// TIA Portal V17 program export: 3 tag tables, 0 data types, 10 data blocks, 17 code blocks (in call order from the OBs), 11 instance data blocks

VAR_GLOBAL   // PLC tag table "ALARMES"
   ALM0 AT %MW100 : Word;   // ALARMES MB-01
   ALM2 AT %MW102 : Word;   // ALARMES MB-02
   ALM4 AT %MW104 : Word;   // ALARMES MB-03
   ALM6 AT %MW106 : Word;   // ALARMES MB-04
   ALM8 AT %MW108 : Word;   // ALARMES LIT_001
   ALM10 AT %MW110 : Word;   // ALARMES PCM-EEE
   ALM12 AT %MW112 : Word;   // ALARMES QGBT
   ALM14 AT %MW114 : Word;   // ALARMES CHAVE DE NIVEL
   ALM16 AT %MW116 : Word;   // ALARMES PCE-EEE
END_VAR

VAR_GLOBAL   // PLC tag table "Default tag table"
   System_Byte AT %MB1 : Byte;
   FirstScan AT %M1.0 : Bool;
   DiagStatusUpdate AT %M1.1 : Bool;
   AlwaysTRUE AT %M1.2 : Bool;
   AlwaysFALSE AT %M1.3 : Bool;
   Clock_Byte AT %MB0 : Byte;
   Clock_10Hz AT %M0.0 : Bool;
   Clock_5Hz AT %M0.1 : Bool;
   "Clock_2.5Hz" AT %M0.2 : Bool;
   Clock_2Hz AT %M0.3 : Bool;
   "Clock_1.25Hz" AT %M0.4 : Bool;
   Clock_1Hz AT %M0.5 : Bool;
   "Clock_0.625Hz" AT %M0.6 : Bool;
   "Clock_0.5Hz" AT %M0.7 : Bool;
   Tag_3 AT %M50.0 : Bool;
   bloqueio_provisorio AT %M2.0 : Bool;
   pause AT %M2.1 : Bool;
   bloqueio_provisorio_1 AT %M2.2 : Bool;
   Tag_4 AT %M83.0 : Bool;
   CON_MOD AT %MW80 : Int;
   INI AT %M82.0 : Bool;
END_VAR

VAR_GLOBAL   // PLC tag table "IO"
   PCM_EEE_EMER AT %I0.0 : Bool;   // PCM-E-CF-01-04 BOTAO DE EMERGENCIA - ATUADO
   PCM_EEE_K27 AT %I0.1 : Bool;   // PCM-E-CF-01-04 RELE DE PROTECAO FUNCAO 27 - ATUADO
   PCM_EEE_DJL AT %I0.2 : Bool;   // PCM-E-CF-01-04 DISJUNTOR GERAL STATUS - LIGADO
   PCM_EEE_DJD AT %I0.3 : Bool;   // PCM-E-CF-01-04 DISJUNTOR GERAL STATUS - DESLIGADO
   PCM_EEE_DJYFAL AT %I0.4 : Bool;   // PCM-E-CF-01-04 DISJUNTOR GERAL STATUS - FALHA
   PCM_EEE_DJFG AT %I0.5 : Bool;   // PCM-E-CF-01-04 FALHA GERAL ATUADO
   PCM_EEE_TR01_KA3 AT %I0.6 : Bool;   // PCM-E-CF-01-04 TRANSFORMADOR -TR-01 ALARME TEMP 150°
   PCM_EEE_TR01_KA4 AT %I0.7 : Bool;   // PCM-E-CF-01-04 TRANSFORMADOR -TR-01 ALARME TEMP 155°
   PCM_EEE_TR01_KA5 AT %I1.0 : Bool;   // PCM-E-CF-01-04 TRANSFORMADOR -TR-01 FALHA PROTECAO
   PCM_EEE_INTRU AT %I1.1 : Bool;   // PCM-E-CF-01-04 INTRUSAO NO PAINEL (COLUNA 01~04)
   MB_01_FF AT %I1.2 : Bool;   // MB-01 FALTA DE FASE
   MB_01_MMNT AT %I1.3 : Bool;   // MB-01 MODO MANUTENCAO
   MB_01_ML AT %I1.4 : Bool;   // MB-01 MODO LOCAL
   MB_01_MA AT %I1.5 : Bool;   // MB-01 MODO AUTOMATICO
   MB_01_MN AT %I1.6 : Bool;   // MB-01 MODO NORMAL
   MB_01_HMNT AT %I1.7 : Bool;   // MB-01 HABILITA MANUTENCAO
   MB_01_BL AT %I2.0 : Bool;   // MB-01 BOMBA LIGADA
   MB_01_DINV AT %I2.1 : Bool;   // MB-01 DEFEITO NO INVERSOR
   MB_01_DMB AT %I2.2 : Bool;   // MB-01 DEFEITO NA BOMBA
   MB_01_RST AT %I2.3 : Bool;   // MB-01 RESET
   MB_01_INTRU AT %I2.4 : Bool;   // MB-01 INTRUSAO NO PAINEL
   MB_01_EMER AT %I2.5 : Bool;   // MB-01 EMERGENCIA
   MB_02_FF AT %I2.6 : Bool;   // MB-02 FALTA DE FASE
   MB_02_MMNT AT %I2.7 : Bool;   // MB-02 MODO MANUTENCAO
   MB_02_ML AT %I3.0 : Bool;   // MB-02 MODO LOCAL
   MB_02_MA AT %I3.1 : Bool;   // MB-02 MODO AUTOMATICO
   MB_02_MN AT %I3.2 : Bool;   // MB-02 MODO NORMAL
   MB_02_HMNT AT %I3.3 : Bool;   // MB-02 HABILITA MANUTENCAO
   MB_02_BL AT %I3.4 : Bool;   // MB-02 BOMBA LIGADA
   MB_02_DINV AT %I3.5 : Bool;   // MB-02 DEFEITO NO INVERSOR
   MB_02_DMB AT %I3.6 : Bool;   // MB-02 DEFEITO NA BOMBA
   MB_02_RST AT %I3.7 : Bool;   // MB-02 RESET
   MB_02_INTRU AT %I4.0 : Bool;   // MB-02 INTRUSAO NO PAINEL
   MB_02_EMER AT %I4.1 : Bool;   // MB-02 EMERGENCIA
   MB_03_FF AT %I4.2 : Bool;   // MB-03 FALTA DE FASE
   MB_03_MMNT AT %I4.3 : Bool;   // MB-03 MODO MANUTENCAO
   MB_03_ML AT %I4.4 : Bool;   // MB-03 MODO LOCAL
   MB_03_MA AT %I4.5 : Bool;   // MB-03 MODO AUTOMATICO
   MB_03_MN AT %I4.6 : Bool;   // MB-03 MODO NORMAL
   MB_03_HMNT AT %I4.7 : Bool;   // MB-03 HABILITA MANUTENCAO
   MB_03_BL AT %I5.0 : Bool;   // MB-03 BOMBA LIGADA
   MB_03_DINV AT %I5.1 : Bool;   // MB-03 DEFEITO NO INVERSOR
   MB_03_DMB AT %I5.2 : Bool;   // MB-03 DEFEITO NA BOMBA
   MB_03_RST AT %I5.3 : Bool;   // MB-03 RESET
   MB_03_INTRU AT %I5.4 : Bool;   // MB-03 INTRUSAO NO PAINEL
   MB_03_EMER AT %I5.5 : Bool;   // MB-03EMERGENCIA
   MB_04_FF AT %I5.6 : Bool;   // MB-04 FALTA DE FASE
   MB_04_MMNT AT %I5.7 : Bool;   // MB-04 MODO MANUTENCAO
   MB_04_ML AT %I6.0 : Bool;   // MB-04 MODO LOCAL
   MB_04_MA AT %I6.1 : Bool;   // MB-04 MODO AUTOMATICO
   MB_04_MN AT %I6.2 : Bool;   // MB-04 MODO NORMAL
   MB_04_HMNT AT %I6.3 : Bool;   // MB-04 HABILITA MANUTENCAO
   MB_04_BL AT %I6.4 : Bool;   // MB-04 BOMBA LIGADA
   MB_04_DINV AT %I6.5 : Bool;   // MB-04 DEFEITO NO INVERSOR
   MB_04_DMB AT %I6.6 : Bool;   // MB-04 DEFEITO NA BOMBA
   MB_04_RST AT %I6.7 : Bool;   // MB-04 RESET
   MB_04_INTRU AT %I7.0 : Bool;   // MB-04 INTRUSAO NO PAINEL
   MB_04_EMER AT %I7.1 : Bool;   // MB-04 EMERGENCIA
   QGBT_EMER AT %I7.2 : Bool;   // QGBT-AUX-01 BOTAO DE EMERGENCIA ATUADO
   QGBT_K27 AT %I7.3 : Bool;   // QGBT-AUX-01 RELE DE PROTECAO FUNCAO 27/59 ATUADO
   QGBT_DISJ_LIG AT %I7.4 : Bool;   // QGBT-AUX-01 DISJUNTOR GERAL STATUS - LIGADO
   QGBT_DISJ_DESLIG AT %I7.5 : Bool;   // QGBT-AUX-01 DISJUNTOR GERAL STATUS - DESLIGADO
   QGBT_DISJ_YFAL AT %I7.6 : Bool;   // QGBT-AUX-01 DISJUNTOR GERAL FALHA - TRIP
   QGBT_INTRU AT %I7.7 : Bool;   // QGBT-AUX-01 INTRUSAO NO PAINEL
   KI165 AT %I8.0 : Bool;   // RESERVA
   KI166 AT %I8.1 : Bool;   // RESERVA
   KI167 AT %I8.2 : Bool;   // RESERVA
   KI168 AT %I8.3 : Bool;   // RESERVA
   KI169 AT %I8.4 : Bool;   // RESERVA
   KI170 AT %I8.5 : Bool;   // RESERVA
   KI171 AT %I8.6 : Bool;   // RESERVA
   KI172 AT %I8.7 : Bool;   // RESERVA
   LSL_001 AT %I9.0 : Bool;   // CHAVE DE NIVEL -LSL-001
   LSH_001 AT %I9.1 : Bool;   // CHAVE DE NIVEL -LSH-001
   LSL_002 AT %I9.2 : Bool;   // CHAVE DE NIVEL -LSL-002
   LSH_002 AT %I9.3 : Bool;   // CHAVE DE NIVEL -LSH-002
   PCE_EEE_INTRU AT %I9.4 : Bool;   // INTRUSAO NO PAINEL
   PCE_EEE_UPS_ALM AT %I9.5 : Bool;   // UPS EM ALARME FALHA NA BATERIA
   PCE_EEE_UPS_FE AT %I9.6 : Bool;   // UPS EM OPERACAO FALTA DE ENERGIA
   PCE_EEE_UPS_CHAR AT %I9.7 : Bool;   // UPS EM ALARME BATERIA CARREGADA
   MB_01_SH AT %Q0.0 : Bool;   // MB-01 SOLICITACAO HIDRAULICA
   MB_01_PH AT %Q0.1 : Bool;   // MB-01 PROTECAO HIDRAULICA
   MB_01_INTV AT %Q0.2 : Bool;   // MB-01 INTERVALO (COM)
   MB_01_RR AT %Q0.3 : Bool;   // MB-01 RESET REMOTO
   MB_01_INTVS AT %Q0.4 : Bool;   // MB-01 INTERVALO SINAL
   MB_02_SH AT %Q0.5 : Bool;   // MB-02 SOLICITACAO HIDRAULICA
   MB_02_PH AT %Q0.6 : Bool;   // MB-02 PROTECAO HIDRAULICA
   MB_02_INTV AT %Q0.7 : Bool;   // MB-02 INTERVALO (COM)
   MB_02_RR AT %Q1.0 : Bool;   // MB-02 RESET REMOTO
   MB_02_INTVS AT %Q1.1 : Bool;   // MB-02 INTERVALO SINAL
   MB_03_SH AT %Q1.2 : Bool;   // MB-03 SOLICITACAO HIDRAULICA
   MB_03_PH AT %Q1.3 : Bool;   // MB-03 PROTECAO HIDRAULICA
   MB_03_INTV AT %Q1.4 : Bool;   // MB-03 INTERVALO (COM)
   MB_03_RR AT %Q1.5 : Bool;   // MB-03 RESET REMOTO
   MB_03_INTVS AT %Q1.6 : Bool;   // MB-03 INTERVALO SINAL
   MB_04_SH AT %Q1.7 : Bool;   // MB-04 SOLICITACAO HIDRAULICA
   LIT_001 AT %IW10 : Int;   // -LIT-001 TRANSMISSOR DE NIVEL TANQUE (TIPO RADAR)
   MB_01_REF_VEL AT %IW12 : Int;   // REFERENCIA DE VELOCIDADE INVERSOR DE FREQUENCIA BOMBA 01
   MB_02_REF_VEL AT %IW14 : Int;   // REFERENCIA DE VELOCIDADE INVERSOR DE FREQUENCIA BOMBA 02
   MB_03_REF_VEL AT %IW16 : Int;   // REFERENCIA DE VELOCIDADE INVERSOR DE FREQUENCIA BOMBA 03
   MB_04_REF_VEL AT %IW18 : Int;   // REFERENCIA DE VELOCIDADE INVERSOR DE FREQUENCIA BOMBA 04
   FB6 AT %IW20 : Int;   // RESERVA
   FB7 AT %IW22 : Int;   // RESERVA
   FB8 AT %IW24 : Int;   // RESERVA
   FB9 AT %IW26 : Int;   // RESERVA
   FB10 AT %IW28 : Int;   // RESERVA
   FB11 AT %IW30 : Int;   // RESERVA
   FB12 AT %IW32 : Int;   // RESERVA
   FB13 AT %IW34 : Int;   // RESERVA
   FB14 AT %IW36 : Int;   // RESERVA
   FB15 AT %IW38 : Int;   // RESERVA
   FB16 AT %IW40 : Int;   // RESERVA
   MB_01_VEL AT %QW4 : Int;   // SETPOINT INVERSOR DE FREQUENCIA BOMBA 01
   MB_02_VEL AT %QW6 : Int;   // SETPOINT INVERSOR DE FREQUENCIA BOMBA 02
   MB_03_VEL AT %QW8 : Int;   // SETPOINT INVERSOR DE FREQUENCIA BOMBA 03
   MB_04_VEL AT %QW10 : Int;   // SETPOINT INVERSOR DE FREQUENCIA BOMBA 04
   F25 AT %QW12 : Int;   // RESERVA
   F26 AT %QW14 : Int;   // RESERVA
   F27 AT %QW16 : Int;   // RESERVA
   F28 AT %QW18 : Int;   // RESERVA
   MB_04_PH AT %Q2.0 : Bool;   // MB-04 PROTECAO HIDRAULICA
   MB_04_INTV AT %Q2.1 : Bool;   // MB-04 INTERVALO (COM)
   MB_04_RR AT %Q2.2 : Bool;   // MB-04 RESET REMOTO
   MB_04_INTVS AT %Q2.3 : Bool;   // MB-04 INTERVALO SINAL
   KO21 AT %Q2.4 : Bool;   // RESERVA
   KO22 AT %Q2.5 : Bool;   // RESERVA
   KO23 AT %Q2.6 : Bool;   // RESERVA
   KO24 AT %Q2.7 : Bool;   // RESERVA
   KO25 AT %Q3.0 : Bool;   // RESERVA
   KO26 AT %Q3.1 : Bool;   // RESERVA
   KO27 AT %Q3.2 : Bool;   // RESERVA
   KO28 AT %Q3.3 : Bool;   // RESERVA
   KO29 AT %Q3.4 : Bool;   // RESERVA
   KO30 AT %Q3.5 : Bool;   // RESERVA
   KO31 AT %Q3.6 : Bool;   // RESERVA
   KO32 AT %Q3.7 : Bool;   // RESERVA
END_VAR

DATA_BLOCK "ALARMES"   // DB301
{ S7_Optimized_Access := 'TRUE' }
VERSION : 0.1
// stored: AutoNumber false, DBAccessibleFromOPCUA true, IsOnlyStoredInLoadMemory false, IsRetainMemResEnabled false, IsWriteProtectedInAS false, MemoryReserve 100
   VAR
      "CCM-02-EA-P100-YFC" : Bool;   // Falha de comunicação com medidor do CCM1
      "CCM-02-EB-P100-YFC" : Bool;   // Falha de comunicação com medidor do CCM2
      "LIT_001-YHH" : Bool;   // Alarme de nível muito alto do tanque água bruta
      "LIT_001-YH" : Bool;   // Alarme de nível alto do tanque água bruta
      "LIT_001-YL" : Bool;   // Alarme de nível baixo do tanque água bruta
      "LIT_001-YLL" : Bool;   // Alarme de nível muito baixo do tanque água bruta
      "LIT_001-YFS" : Bool;   // Transmissor de nível do tanque água bruta com falha de sinal
      "LIT_001-YHHH" : Bool;   // Alarme de nível muito alto - desliga CAB e lavagem peneira
      "CAB-PT-015-YH" : Bool;
      "CAB-PT-015-YFS" : Bool;
      "MB-03-YIP" : Bool;   // MB-03 com intervalo entre partidas
      "MB-02-YIP" : Bool;   // MB-02 com intervalo entre partidas
      "MB-01-YIP" : Bool;   // MB-01 com intervalo entre partidas
   END_VAR
BEGIN
END_DATA_BLOCK

DATA_BLOCK "COMANDOS"   // DB303
{ S7_Optimized_Access := 'FALSE' }
VERSION : 0.1
// stored: AutoNumber false, DBAccessibleFromOPCUA true, IsOnlyStoredInLoadMemory false, IsWriteProtectedInAS false
   VAR RETAIN
      "MB-01-HS9" : Bool := false;   // Comando disponível
      "MB-01-HS10" : Bool := false;   // Comando disponível
      "MB-01-HS11" : Bool;   // Comando disponível
      "MB-01-HS12" : Bool;   // Comando disponível
      "MB-01-HS13" : Bool;   // Comando disponível
      "MB-01-HS14" : Bool;   // Comando disponível
      "MB-01-HS15" : Bool;   // Comando disponível
      "MB-01-HS16" : Bool;   // Comando disponível
      "MB-01-HS1" : Bool := true;   // Comando manual/automático
      "MB-01-HS2" : Bool := false;   // Comando liga
      "MB-01-HS3" : Bool := false;   // Comando desliga
      "MB-01-HS4" : Bool := false;   // Comando reset falha
      "MB-01-HS5" : Bool := false;   // Comando reset tempo de operação
      "MB-01-HS6" : Bool;
      "MB-01-HS7" : Bool := false;   // Comando habilita bloqueio
      "MB-01-HS8" : Bool := false;   // Comando disponível
      "MB-02-HS9" : Bool := false;   // Comando disponível
      "MB-02-HS10" : Bool := false;   // Comando disponível
      "MB-02-HS11" : Bool;   // Comando disponível
      "MB-02-HS12" : Bool;   // Comando disponível
      "MB-02-HS13" : Bool;   // Comando disponível
      "MB-02-HS14" : Bool;   // Comando disponível
      "MB-02-HS15" : Bool;   // Comando disponível
      "MB-02-HS16" : Bool;   // Comando disponível
      "MB-02-HS1" : Bool := true;   // Comando manual/automático
      "MB-02-HS2" : Bool := false;   // Comando liga
      "MB-02-HS3" : Bool := false;   // Comando desliga
      "MB-02-HS4" : Bool := false;   // Comando reset falha
      "MB-02-HS5" : Bool := false;   // Comando reset tempo de operação
      "MB-02-HS6" : Bool;
      "MB-02-HS7" : Bool := false;   // Comando habilita bloqueio
      "MB-02-HS8" : Bool := false;   // Comando disponível
      "MB-03-HS9" : Bool := false;   // Comando disponível
      "MB-03-HS10" : Bool := false;   // Comando disponível
      "MB-03-HS11" : Bool;   // Comando disponível
      "MB-03-HS12" : Bool;   // Comando disponível
      "MB-03-HS13" : Bool;   // Comando disponível
      "MB-03-HS14" : Bool;   // Comando disponível
      "MB-03-HS15" : Bool;   // Comando disponível
      "MB-03-HS16" : Bool;   // Comando disponível
      "MB-03-HS1" : Bool := true;   // Comando manual/automático
      "MB-03-HS2" : Bool := false;   // Comando liga
      "MB-03-HS3" : Bool := false;   // Comando desliga
      "MB-03-HS4" : Bool := false;   // Comando reset falha
      "MB-03-HS5" : Bool := false;   // Comando reset tempo de operação
      "MB-03-HS6" : Bool;
      "MB-03-HS7" : Bool := false;   // Comando habilita bloqueio
      "MB-03-HS8" : Bool := false;   // Comando disponível
      "MB-04-HS9" : Bool := false;   // Comando disponível
      "MB-04-HS10" : Bool := false;   // Comando disponível
      "MB-04-HS11" : Bool;   // Comando disponível
      "MB-04-HS12" : Bool;   // Comando disponível
      "MB-04-HS13" : Bool;   // Comando disponível
      "MB-04-HS14" : Bool;   // Comando disponível
      "MB-04-HS15" : Bool;   // Comando disponível
      "MB-04-HS16" : Bool;   // Comando disponível
      "MB-04-HS1" : Bool := false;   // Comando manual/automático
      "MB-04-HS2" : Bool := false;   // Comando liga
      "MB-04-HS3" : Bool := false;   // Comando desliga
      "MB-04-HS4" : Bool := false;   // Comando reset falha
      "MB-04-HS5" : Bool := false;   // Comando reset tempo de operação
      "MB-04-HS6" : Bool;
      "MB-04-HS7" : Bool := false;   // Comando habilita bloqueio
      "MB-04-HS8" : Bool := false;   // Comando disponível
      "LIT_001-HS9" : Bool;   // Comando disponível
      "LIT_001-HS10" : Bool;   // Comando disponível
      "LIT_001-HS11" : Bool;   // Comando disponível
      "LIT_001-HS12" : Bool;   // Comando disponível
      "LIT_001-HS13" : Bool;   // Comando disponível
      "LIT_001-HS14" : Bool;   // Comando disponível
      "LIT_001-HS15" : Bool;   // Comando disponível
      "LIT_001-HS16" : Bool;   // Comando disponível
      "LIT_001-HSHH" : Bool;   // Inibe alarme muito alto montante peneira 1
      "LIT_001-HSH" : Bool;   // Inibe alarme nível alto montante peneira 1
      "LIT_001-HSL" : Bool;   // Inibe alarme nível baixo montante peneira 1
      "LIT_001-HSLL" : Bool;   // Inibe alarme nível muito baixo montante peneira 1
      "LIT_001-HSM" : Bool;   // Habilita valor manual para medidor
      "LIT_001-HS6" : Bool;   // Comando disponível
      "LIT_001-HS7" : Bool;   // Comando disponível
      "LIT_001-HS8" : Bool;   // Comando disponível
      "PID-TA3-HI" : Bool;   // Habilita integrall PID tanque de aeração
      "PID-EEEB-HD" : Bool;   // Habilita derivativo PID tanque de aeração
      "PID-EEEB-HP" : Bool;   // Habilita proporcional PID tanque de aeração
      "PID-EEEB-HI" : Bool;   // Habilita integrall PID tanque de aeração
      "PID-TA5-HD" : Bool;   // Habilita derivativo PID tanque de aeração
      "PID-TA5-HP" : Bool;   // Habilita proporcional PID tanque de aeração
      "PID-TA5-HI" : Bool;   // Habilita integrall PID tanque de aeração
      "PID-TA1-HM" : Bool;   // Habilita valor manual para saída
      "PID-TA1-HD" : Bool;   // Habilita derivativo PID tanque de aeração
      "PID-TA1-HP" : Bool;   // Habilita proporcional PID tanque de aeração
      "PID-TA1-HI" : Bool;   // Habilita integrall PID tanque de aeração
      "PID-TA2-HD" : Bool;   // Habilita derivativo PID tanque de aeração
      "PID-TA2-HP" : Bool;   // Habilita proporcional PID tanque de aeração
      "PID-TA2-HI" : Bool;   // Habilita integrall PID tanque de aeração
      "PID-TA3-HD" : Bool;   // Habilita derivativo PID tanque de aeração
      "PID-TA3-HP" : Bool;   // Habilita proporcional PID tanque de aeração
      "PID-TA2-HM" : Bool;   // Habilita valor manual para saída
      "PID-TA3-HM" : Bool;   // Habilita valor manual para saída
      "PID-EEEB-HM" : Bool;   // Habilita valor manual para saída
      "PID-TA5-HM" : Bool;   // Habilita valor manual para saída
   END_VAR
BEGIN
END_DATA_BLOCK

DATA_BLOCK "DIVERSOS"   // DB1
{ S7_Optimized_Access := 'TRUE' }
VERSION : 0.1
// stored: AutoNumber false, DBAccessibleFromOPCUA true, IsOnlyStoredInLoadMemory false, IsRetainMemResEnabled false, IsWriteProtectedInAS false, MemoryReserve 100
   VAR
      T1S : Bool;   // PULSO A CADA 1 SEGUNDO
      AUX_T1S : Bool;   // PULSO A CADA 1 SEGUNDO
      QTDE_PULSO : DInt := 200;
      ForcePulso : Bool;
      N_L00P : Int;
      Aux_N_LOOP : Int;
      Looping : Int := 0;
      TMR : Array[0..10] of IEC_TIMER;
      P1S { S7_SetPoint := 'True'} : Bool;   // Pulso de 1 segundo
      "MB-01-SP" : Bool;   // Solicitação partida de bomba
      "MB-02-SP" : Bool;   // Solicitação partida de bomba
      "MB-03-SP" : Bool;   // Solicitação partida de bomba
      "MB-04-SP" : Bool;   // Solicitação partida de bomba
   END_VAR
BEGIN
END_DATA_BLOCK

DATA_BLOCK "Digitais"   // DB300
{ S7_Optimized_Access := 'FALSE' }
VERSION : 0.1
// stored: AutoNumber false, DBAccessibleFromOPCUA true, IsOnlyStoredInLoadMemory false, IsWriteProtectedInAS false
   VAR RETAIN
      "MB-01-YSH" : Bool;   // Elevatoria principal 1 ligado
      "MB-01-YR" : Bool;   // Elevatoria principal 1 remoto
      "MB-01-YF" : Bool;   // Elevatoria principal 1 falha
      "MB-01-YFF" : Bool;   // Elevatoria principal 1 falta de fase
      "MB-01-MM" : Bool;   // Elevatoria principal 1 modo manutenção
      "MB-01-MA" : Bool;   // Elevatoria principal 1 modo automatico
      "MB-01-EMER" : Bool;   // Elevatoria principal 1 emergencia
      "MB-01-MN" : Bool;   // Elevatoria principal 1 modo normal
      "MB-01-ML" : Bool;   // Elevatoria principal 1 modo local
      "MB-01-YFI" : Bool;   // Elevatoria principal 1 com falha no inversor
      "MB-01-YFA" : Bool;   // Elevatoria principal 1 com falha no acionamento
      "MB-01-YPTA" : Bool;   // Elevatoria principal 1 com proteção térmica atuada
      "MB-01-HM" : Bool;   // Elevatoria principal 1 habilita manutenção
      "MB-01-RST" : Bool;   // Elevatoria principal 1 reset
      "MB-01-INTRU" : Bool;   // Elevatoria principal 1 intrusão no painel
      "MB-01-YFB" : Bool;   // Elevatoria principal 1 defeito na bomba
      "MB-02-YSH" : Bool;   // Elevatoria principal 2 ligado
      "MB-02-YR" : Bool;   // Elevatoria principal 2 remoto
      "MB-02-YF" : Bool;   // Elevatoria principal 2 falha
      "MB-02-YFF" : Bool;   // Elevatoria principal 2 falta de fase
      "MB-02-MM" : Bool;   // Elevatoria principal 2 modo manutenção
      "MB-02-MA" : Bool;   // Elevatoria principal 2 modo automatico
      "MB-02-EMER" : Bool;   // Elevatoria principal 2 emergencia
      "MB-02-MN" : Bool;   // Elevatoria principal 2 modo normal
      "MB-02-ML" : Bool;   // Elevatoria principal 2 modo local
      "MB-02-YFI" : Bool;   // Elevatoria principal 2 com falha no inversor
      "MB-02-YFA" : Bool;   // Elevatoria principal 2 com falha no acionamento
      "MB-02-YPTA" : Bool;   // Elevatoria principal 2 com proteção térmica atuada
      "MB-02-HM" : Bool;   // Elevatoria principal 2 habilita manutenção
      "MB-02-RST" : Bool;   // Elevatoria principal 2 reset
      "MB-02-INTRU" : Bool;   // Elevatoria principal 2 intrusão no painel
      "MB-02-YFB" : Bool;   // Elevatoria principal 2 defeito na bomba
      "MB-03-YSH" : Bool;   // Elevatoria principal 3 ligado
      "MB-03-YR" : Bool;   // Elevatoria principal 3 remoto
      "MB-03-YF" : Bool;   // Elevatoria principal 3 falha
      "MB-03-YFF" : Bool;   // Elevatoria principal 3 falta de fase
      "MB-03-MM" : Bool;   // Elevatoria principal 3 modo manutenção
      "MB-03-MA" : Bool;   // Elevatoria principal 3 modo automatico
      "MB-03-EMER" : Bool;   // Elevatoria principal 3 emergencia
      "MB-03-MN" : Bool;   // Elevatoria principal 3 modo normal
      "MB-03-ML" : Bool;   // Elevatoria principal 3 modo local
      "MB-03-YFI" : Bool;   // Elevatoria principal 3 com falha no inversor
      "MB-03-YFA" : Bool;   // Elevatoria principal 3 com falha no acionamento
      "MB-03-YPTA" : Bool;   // Elevatoria principal 3 com proteção térmica atuada
      "MB-03-HM" : Bool;   // Elevatoria principal 3 habilita manutenção
      "MB-03-RST" : Bool;   // Elevatoria principal 3 reset
      "MB-03-INTRU" : Bool;   // Elevatoria principal 3 intrusão no painel
      "MB-03-YFB" : Bool;   // Elevatoria principal 3 defeito na bomba
      "MB-04-YSH" : Bool;   // Elevatoria principal 4 ligado
      "MB-04-YR" : Bool;   // Elevatoria principal 4 remoto
      "MB-04-YF" : Bool;   // Elevatoria principal 4 falha
      "MB-04-YFF" : Bool;   // Elevatoria principal 4 falta de fase
      "MB-04-MM" : Bool;   // Elevatoria principal 4 modo manutenção
      "MB-04-MA" : Bool;   // Elevatoria principal 4 modo automatico
      "MB-04-EMER" : Bool;   // Elevatoria principal 4 emergencia
      "MB-04-MN" : Bool;   // Elevatoria principal 4 modo normal
      "MB-04-ML" : Bool;   // Elevatoria principal 4 modo local
      "MB-04-YFI" : Bool;   // Elevatoria principal 4 com falha no inversor
      "MB-04-YFA" : Bool;   // Elevatoria principal 4 com falha no acionamento
      "MB-04-YPTA" : Bool;   // Elevatoria principal 4 com proteção térmica atuada
      "MB-04-HM" : Bool;   // Elevatoria principal 4 habilita manutenção
      "MB-04-RST" : Bool;   // Elevatoria principal 4 reset
      "MB-04-INTRU" : Bool;   // Elevatoria principal 4 intrusão no painel
      "MB-04-YFB" : Bool;   // Elevatoria principal 4 defeito na bomba
      "LIT_001-AL8" : Bool;   // Disponível para alarme
      "LIT_001-AL9" : Bool;   // Disponível para alarme
      "LIT_001-AL10" : Bool;   // Disponível para alarme
      "LIT_001-AL11" : Bool;   // Disponível para alarme
      "LIT_001-AL12" : Bool;   // Disponível para alarme
      "LIT_001-AL13" : Bool;   // Disponível para alarme
      "LIT_001-AL14" : Bool;   // Disponível para alarme
      "LIT_001-AL15" : Bool;   // Disponível para alarme
      "LIT_001-YHH" : Bool;   // Alarme de nível muito alto do tanque
      "LIT_001-YH" : Bool;   // Alarme de nível alto do tanque
      "LIT_001-YL" : Bool;   // Alarme de nível baixo do tanque
      "LIT_001-YLL" : Bool;   // Alarme de nível muito baixo do tanque
      "LIT_001-YFS" : Bool;   // Transmissor de nível do tanque com falha de sinal
      "LIT_001-AL5" : Bool;   // Disponível para alarme
      "LIT_001-AL6" : Bool;   // Disponível para alarme
      "LIT_001-AL7" : Bool;   // Disponível para alarme
      PCM_EEE_EMER : Bool;   // PCM-E-CF-01-04 BOTAO DE EMERGENCIA - ATUADO
      PCM_EEE_K27 : Bool;   // PCM-E-CF-01-04 RELE DE PROTECAO FUNCAO 27 - ATUADO
      PCM_EEE_DISJ_LIG : Bool;   // PCM-E-CF-01-04 DISJUNTOR GERAL STATUS - LIGADO
      PCM_EEE_DISJ_DESLIG : Bool;   // PCM-E-CF-01-04 DISJUNTOR GERAL STATUS - DESLIGADO
      PCM_EEE_DISJ_YFAL : Bool;   // PCM-E-CF-01-04 DISJUNTOR GERAL STATUS - FALHA
      PCM_EEE_DISJ_FAL_GR : Bool;   // PCM-E-CF-01-04 FALHA GERAL ATUADO
      PCM_EEE_TR01_KA3 : Bool;   // PCM-E-CF-01-04 TRANSFORMADOR -TR-01 ALARME TEMP 150°
      PCM_EEE_TR01_KA4 : Bool;   // PCM-E-CF-01-04 TRANSFORMADOR -TR-01 ALARME TEMP 155°
      PCM_EEE_TR01_KA5 : Bool;   // PCM-E-CF-01-04 TRANSFORMADOR -TR-01 FALHA PROTECAO
      PCM_EEE_INTRU : Bool;   // PCM-E-CF-01-04 INTRUSAO NO PAINEL (COLUNA 01~04)
      PCM_EEE_RSERVA_0 : Bool;   // PCM-E-CF-01-04 BIT RESERVA DA WORD
      PCM_EEE_RSERVA_1 : Bool;   // PCM-E-CF-01-04 BIT RESERVA DA WORD
      PCM_EEE_RSERVA_2 : Bool;   // PCM-E-CF-01-04 BIT RESERVA DA WORD
      PCM_EEE_RSERVA_3 : Bool;   // PCM-E-CF-01-04 BIT RESERVA DA WORD
      PCM_EEE_RSERVA_4 : Bool;   // PCM-E-CF-01-04 BIT RESERVA DA WORD
      PCM_EEE_RSERVA_5 : Bool;   // PCM-E-CF-01-04 BIT RESERVA DA WORD
      QGBT_EMER : Bool;   // QGBT-AUX-01 BOTAO DE EMERGENCIA ATUADO
      QGBT_K27 : Bool;   // QGBT-AUX-01 RELE DE PROTECAO FUNCAO 27/59 ATUADO
      QGBT_DJL : Bool;   // QGBT-AUX-01 DISJUNTOR GERAL STATUS - LIGADO
      QGBT_DJD : Bool;   // QGBT-AUX-01 DISJUNTOR GERAL STATUS - DESLIGADO
      QGBT_DJYFAL : Bool;   // QGBT-AUX-01 DISJUNTOR GERAL FALHA - TRIP
      QGBT_INTRU : Bool;   // QGBT-AUX-01 INTRUSAO NO PAINEL
      QGBT_RESERVA_0 : Bool;   // QGBT-AUX-01 BIT RESERVA DA WORD
      QGBT_RESERVA_1 : Bool;   // QGBT-AUX-01 BIT RESERVA DA WORD
      QGBT_RESERVA_2 : Bool;   // QGBT-AUX-01 BIT RESERVA DA WORD
      QGBT_RESERVA_3 : Bool;   // QGBT-AUX-01 BIT RESERVA DA WORD
      QGBT_RESERVA_4 : Bool;   // QGBT-AUX-01 BIT RESERVA DA WORD
      QGBT_RESERVA_5 : Bool;   // QGBT-AUX-01 BIT RESERVA DA WORD
      QGBT_RESERVA_6 : Bool;   // QGBT-AUX-01 BIT RESERVA DA WORD
      QGBT_RESERVA_7 : Bool;   // QGBT-AUX-01 BIT RESERVA DA WORD
      QGBT_RESERVA_8 : Bool;   // QGBT-AUX-01 BIT RESERVA DA WORD
      QGBT_RESERVA_9 : Bool;   // QGBT-AUX-01 BIT RESERVA DA WORD
      LSL_001 : Bool;   // CHAVE DE NIVEL -LSL-001
      LSH_001 : Bool;   // CHAVE DE NIVEL -LSH-001
      LSL_002 : Bool;   // CHAVE DE NIVEL -LSL-002
      LSH_002 : Bool;   // CHAVE DE NIVEL -LSH-002
      LS_RESERVA_0 : Bool;   // CHAVE DE NIVEL - LS BIT RESERVA DA WORD
      LS_RESERVA_1 : Bool;   // CHAVE DE NIVEL - LS BIT RESERVA DA WORD
      LS_RESERVA_2 : Bool;   // CHAVE DE NIVEL - LS BIT RESERVA DA WORD
      LS_RESERVA_3 : Bool;   // CHAVE DE NIVEL - LS BIT RESERVA DA WORD
      LS_RESERVA_4 : Bool;   // CHAVE DE NIVEL - LS BIT RESERVA DA WORD
      LS_RESERVA_5 : Bool;   // CHAVE DE NIVEL - LS BIT RESERVA DA WORD
      LS_RESERVA_6 : Bool;   // CHAVE DE NIVEL - LS BIT RESERVA DA WORD
      LS_RESERVA_7 : Bool;   // CHAVE DE NIVEL - LS BIT RESERVA DA WORD
      LS_RESERVA_8 : Bool;   // CHAVE DE NIVEL - LS BIT RESERVA DA WORD
      LS_RESERVA_9 : Bool;   // CHAVE DE NIVEL - LS BIT RESERVA DA WORD
      LS_RESERVA_10 : Bool;   // CHAVE DE NIVEL - LS BIT RESERVA DA WORD
      LS_RESERVA_11 : Bool;   // CHAVE DE NIVEL - LS BIT RESERVA DA WORD
      PCE_EEE_INTRU : Bool;   // INTRUSAO NO PAINEL
      PCE_EEE_UPS_ALM : Bool;   // UPS EM ALARME FALHA NA BATERIA
      PCE_EEE_UPS_FE : Bool;   // UPS EM OPERACAO FALTA DE ENERGIA
      PCE_EEE_UPS_CHAR : Bool;   // UPS EM ALARME BATERIA CARREGADA
      "PCM-E-CF-01-P100-YFC" : Bool;   // Falha de comunicação com medidor do PCM-E-CF-01
      "QGBT-AUX-01-P100-YFC" : Bool;   // Falha de comunicação com medidor do PCM-E-CF-02
   END_VAR
BEGIN
END_DATA_BLOCK

DATA_BLOCK "PID"   // DB307
{ S7_Optimized_Access := 'FALSE' }
VERSION : 0.1
// stored: AutoNumber false, DBAccessibleFromOPCUA true, IsOnlyStoredInLoadMemory false, IsWriteProtectedInAS false
   VAR RETAIN
      "PID-EEEB-D" : Real;   // Ajuste derivativo PID elevatória de esgoto bruto
      "PID-EEEB-P" : Real;   // Ajuste proporcional PID elevatória de esgoto bruto
      "PID-EEEB-I" : Real;   // Ajuste integral PID elevatória de esgoto bruto
      "PID-EEEB-MIN" : Real;   // Ajuste mínimo PID elevatória de esgoto bruto
      "PID-EEEB-MAX" : Real;   // Ajuste máximo PID elevatória de esgoto bruto
      "PID-EEEB-DB" : Real;   // Banda morta PID elevatória de esgoto bruto
      "PID-EEEB-SPM" : Real;   // Setpoint manual
      "VA-PID-EEEB" : Real;   // Variável atuada PID elevatória de esgoto bruto
      "PID-EEEB-VR" : Real;   // Valor Relativo do PID
      AUX_CALC : Array[0..10] of Real;
   END_VAR
BEGIN
END_DATA_BLOCK

DATA_BLOCK "Redes"   // DB500
{ S7_Optimized_Access := 'FALSE' }
VERSION : 0.1
// stored: AutoNumber false, DBAccessibleFromOPCUA true, IsOnlyStoredInLoadMemory false, IsWriteProtectedInAS false
   VAR
      "CONNECT-MGE-PCM-E-CF-01" { S7_SetPoint := 'True'} : TCON_IP_v4;   // Dados de configuração
      "CONNECT-MGE-QGBT-AUX-01" { S7_SetPoint := 'True'} : TCON_IP_v4;   // Dados de configuração
      "Register-MGE-PCM-E-CF-01" : Array[0..38] of DInt;   // Tabela para receber os dados
      "Register-MGE-QGBT-AUX-01" : Array[0..38] of DInt;   // Tabela para receber os dados
      LADDR_PROFINET : HW_IOSYSTEM := 261;   // Endereço de hardware
      MODE_PROFINET : UInt := 4;   // Modo de operação da funcção
      RET_VAL_PROFINET : Int;   // Terorno de diagnóstico
      ESTADO_PROFINET : Array[0..1023] of Bool;   // Diagnóstico da rede PROFINET
      DONE_MB : Array[0..60] of Bool;   // Sinaliza fim de execução
      BUSY_MB : Array[0..60] of Bool;   // Sinaliza espera
      ERROR_MB : Array[0..60] of Bool;   // Sinaliza erro
      STATUS_MB : Array[0..60] of Word;   // Satus da comunicação
      START_MB : Array[0..60] of Bool;   // Inicia comunicação
      FCOM_MB : Array[0..60] of Bool;   // Falha de comunicação
      HAB_MB : Array[0..60] of Bool;   // Habilita comunicação MODBUS
      INICIA_MB : Bool;   // INICIA CICLO DE COMUNICAÇÃO MODBUS
      INI_AUX_MB : Bool;   // AUXILIAR DE INICIALIZAÇÃO
   END_VAR
BEGIN
   "CONNECT-MGE-PCM-E-CF-01".InterfaceId := 64;
   "CONNECT-MGE-PCM-E-CF-01".ID := 10;
   "CONNECT-MGE-PCM-E-CF-01".ConnectionType := 11;
   "CONNECT-MGE-PCM-E-CF-01".ActiveEstablished := TRUE;
   "CONNECT-MGE-PCM-E-CF-01".RemoteAddress.ADDR[1] := 192;
   "CONNECT-MGE-PCM-E-CF-01".RemoteAddress.ADDR[2] := 168;
   "CONNECT-MGE-PCM-E-CF-01".RemoteAddress.ADDR[3] := 2;
   "CONNECT-MGE-PCM-E-CF-01".RemoteAddress.ADDR[4] := 59;
   "CONNECT-MGE-PCM-E-CF-01".RemotePort := 502;
   "CONNECT-MGE-PCM-E-CF-01".LocalPort := 0;
   "CONNECT-MGE-QGBT-AUX-01".InterfaceId := 64;
   "CONNECT-MGE-QGBT-AUX-01".ID := 10;
   "CONNECT-MGE-QGBT-AUX-01".ConnectionType := 11;
   "CONNECT-MGE-QGBT-AUX-01".ActiveEstablished := TRUE;
   "CONNECT-MGE-QGBT-AUX-01".RemoteAddress.ADDR[1] := 192;
   "CONNECT-MGE-QGBT-AUX-01".RemoteAddress.ADDR[2] := 168;
   "CONNECT-MGE-QGBT-AUX-01".RemoteAddress.ADDR[3] := 2;
   "CONNECT-MGE-QGBT-AUX-01".RemoteAddress.ADDR[4] := 59;
   "CONNECT-MGE-QGBT-AUX-01".RemotePort := 502;
   "CONNECT-MGE-QGBT-AUX-01".LocalPort := 0;
   // "Register-MGE-PCM-E-CF-01"[0] : Tensão (L-N) fase 1
   // "Register-MGE-PCM-E-CF-01"[1] : Tensão (L-L) fase 1-2
   // "Register-MGE-PCM-E-CF-01"[2] : Corrente fase 1
   // "Register-MGE-PCM-E-CF-01"[3] : Cos φ fase 1
   // "Register-MGE-PCM-E-CF-01"[4] : Fator de potencia fase 1
   // "Register-MGE-PCM-E-CF-01"[5] : Potencia ativa fase 1
   // "Register-MGE-PCM-E-CF-01"[6] : Potência reativa fase 1
   // "Register-MGE-PCM-E-CF-01"[7] : Potência aparente fase 1
   // "Register-MGE-PCM-E-CF-01"[8] : THDV fase 1
   // "Register-MGE-PCM-E-CF-01"[9] : THDI fase 1
   // "Register-MGE-PCM-E-CF-01"[10] : Tensão (L-N) fase 2
   // "Register-MGE-PCM-E-CF-01"[11] : Tensão (L-L) fase 2-3
   // "Register-MGE-PCM-E-CF-01"[12] : Corrente fase 2
   // "Register-MGE-PCM-E-CF-01"[13] : Cos φ fase 2
   // "Register-MGE-PCM-E-CF-01"[14] : Fator de potência fase 2
   // "Register-MGE-PCM-E-CF-01"[15] : Potência ativa fase 2
   // "Register-MGE-PCM-E-CF-01"[16] : Potência reativa fase 2
   // "Register-MGE-PCM-E-CF-01"[17] : Potência aparente fase 2
   // "Register-MGE-PCM-E-CF-01"[18] : THDV fase 2
   // "Register-MGE-PCM-E-CF-01"[19] : THDI fase 2
   // "Register-MGE-PCM-E-CF-01"[20] : Tensão (L-N) fase 3
   // "Register-MGE-PCM-E-CF-01"[21] : Tensão (L-L) fase 3-1
   // "Register-MGE-PCM-E-CF-01"[22] : Corrente fase 3
   // "Register-MGE-PCM-E-CF-01"[23] : Cos φ fase 3
   // "Register-MGE-PCM-E-CF-01"[24] : Fator de potência fase 3
   // "Register-MGE-PCM-E-CF-01"[25] : Potência ativa fase 3
   // "Register-MGE-PCM-E-CF-01"[26] : Potência reativa fase 3
   // "Register-MGE-PCM-E-CF-01"[27] : Potência aparente fase 3
   // "Register-MGE-PCM-E-CF-01"[28] : THDV fase 3
   // "Register-MGE-PCM-E-CF-01"[29] : THDI fase 3
   // "Register-MGE-PCM-E-CF-01"[30] : Tensão média (L-N)
   // "Register-MGE-PCM-E-CF-01"[31] : Tensão média (L-L)
   // "Register-MGE-PCM-E-CF-01"[32] : Corrente total
   // "Register-MGE-PCM-E-CF-01"[33] : Fator de potência do sistema
   // "Register-MGE-PCM-E-CF-01"[34] : Potência ativa total
   // "Register-MGE-PCM-E-CF-01"[35] : Potência reativa total
   // "Register-MGE-PCM-E-CF-01"[36] : Potência aparente total
   // "Register-MGE-PCM-E-CF-01"[37] : Frequência do sistema
   // "Register-MGE-PCM-E-CF-01"[38] : Corrente de neutro
   // "Register-MGE-QGBT-AUX-01"[0] : Tensão (L-N) fase 1
   // "Register-MGE-QGBT-AUX-01"[1] : Tensão (L-L) fase 1-2
   // "Register-MGE-QGBT-AUX-01"[2] : Corrente fase 1
   // "Register-MGE-QGBT-AUX-01"[3] : Cos φ fase 1
   // "Register-MGE-QGBT-AUX-01"[4] : Fator de potencia fase 1
   // "Register-MGE-QGBT-AUX-01"[5] : Potencia ativa fase 1
   // "Register-MGE-QGBT-AUX-01"[6] : Potência reativa fase 1
   // "Register-MGE-QGBT-AUX-01"[7] : Potência aparente fase 1
   // "Register-MGE-QGBT-AUX-01"[8] : THDV fase 1
   // "Register-MGE-QGBT-AUX-01"[9] : THDI fase 1
   // "Register-MGE-QGBT-AUX-01"[10] : Tensão (L-N) fase 2
   // "Register-MGE-QGBT-AUX-01"[11] : Tensão (L-L) fase 2-3
   // "Register-MGE-QGBT-AUX-01"[12] : Corrente fase 2
   // "Register-MGE-QGBT-AUX-01"[13] : Cos φ fase 2
   // "Register-MGE-QGBT-AUX-01"[14] : Fator de potência fase 2
   // "Register-MGE-QGBT-AUX-01"[15] : Potência ativa fase 2
   // "Register-MGE-QGBT-AUX-01"[16] : Potência reativa fase 2
   // "Register-MGE-QGBT-AUX-01"[17] : Potência aparente fase 2
   // "Register-MGE-QGBT-AUX-01"[18] : THDV fase 2
   // "Register-MGE-QGBT-AUX-01"[19] : THDI fase 2
   // "Register-MGE-QGBT-AUX-01"[20] : Tensão (L-N) fase 3
   // "Register-MGE-QGBT-AUX-01"[21] : Tensão (L-L) fase 3-1
   // "Register-MGE-QGBT-AUX-01"[22] : Corrente fase 3
   // "Register-MGE-QGBT-AUX-01"[23] : Cos φ fase 3
   // "Register-MGE-QGBT-AUX-01"[24] : Fator de potência fase 3
   // "Register-MGE-QGBT-AUX-01"[25] : Potência ativa fase 3
   // "Register-MGE-QGBT-AUX-01"[26] : Potência reativa fase 3
   // "Register-MGE-QGBT-AUX-01"[27] : Potência aparente fase 3
   // "Register-MGE-QGBT-AUX-01"[28] : THDV fase 3
   // "Register-MGE-QGBT-AUX-01"[29] : THDI fase 3
   // "Register-MGE-QGBT-AUX-01"[30] : Tensão média (L-N)
   // "Register-MGE-QGBT-AUX-01"[31] : Tensão média (L-L)
   // "Register-MGE-QGBT-AUX-01"[32] : Corrente total
   // "Register-MGE-QGBT-AUX-01"[33] : Fator de potência do sistema
   // "Register-MGE-QGBT-AUX-01"[34] : Potência ativa total
   // "Register-MGE-QGBT-AUX-01"[35] : Potência reativa total
   // "Register-MGE-QGBT-AUX-01"[36] : Potência aparente total
   // "Register-MGE-QGBT-AUX-01"[37] : Frequência do sistema
   // "Register-MGE-QGBT-AUX-01"[38] : Corrente de neutro
END_DATA_BLOCK

DATA_BLOCK "SETPOINTS"   // DB305
{ S7_Optimized_Access := 'FALSE' }
VERSION : 0.1
// stored: AutoNumber false, DBAccessibleFromOPCUA true, IsOnlyStoredInLoadMemory false, IsWriteProtectedInAS false
   VAR RETAIN
      "MB-01-SP" : Real := 60.0;   // Setpoint manual elevatoria principal
      "MB-02-SP" : Real := 0.0;   // Setpoint manual elevatoria principal
      "MB-03-SP" : Real := 60.0;   // Setpoint manual elevatoria principal
      "MB-04-SP" : Real := 60.0;   // Setpoint manual elevatoria principal
      "LIT_001-SPHH" : Real := 90.0;   // Setpoint muito alto elevatoria principal
      "LIT_001-SPH" : Real := 70.0;   // Setpoint nível alto elevatoria principal
      "LIT_001-SPL" : Real := 10.0;   // Setpoint nível baixo elevatoria principal
      "LIT_001-SPLL" : Real := 0.0;   // Setpoint nível muito baixo elevatoria principal
      "LIT_001-SPM" : Real := 48.0;   // Habilita valor manual para medidor
      "LIT_001-SPC" : Real := 0.0;   // Setpoint de controle tanque
      "LIT-001-P" : Real := 0.0;
      SP_NVL_MIN : Real := 1.0;   // setpoint nivel minimo do tanque para proteção hidraulica
      "MB-P-SP-DL" : Real := 2.0;   // Setpoint para desligar bomba Principal
      "MB-P-SP-L" : Real := 2.6;   // Setpoint para ligar bomba Principal
      "MB-C1-SP-DL" : Real := 2.35;   // Setpoint para desligar bomba complementar 1
      "MB-C1-SP-L" : Real := 2.9;   // Setpoint para ligar bomba complementar 1
      "MB-C2-SP-DL" : Real := 2.66;   // Setpoint para desligar bomba complementar 2
      "MB-C2-SP-L" : Real := 3.9;   // Setpoint para ligar bomba complementar 2
      "MB-C3-SP-DL" : Real := 0.0;   // Setpoint para desligar bomba complementar 3
      "MB-C3-SP-L" : Real := 0.0;   // Setpoint para ligar bomba complementar 3
   END_VAR
BEGIN
END_DATA_BLOCK

DATA_BLOCK "STATUS"   // DB302
{ S7_Optimized_Access := 'FALSE' }
VERSION : 0.1
// stored: AutoNumber false, DBAccessibleFromOPCUA true, IsOnlyStoredInLoadMemory false, IsWriteProtectedInAS false
   VAR
      "SO-203-06A-YI" : Bool;   // Soprador tanque de aeração intertravado
      "SO-203-06B-YI" : Bool;   // Soprador tanque de aeração intertravado
      "SO-203-06C-YI" : Bool;   // Soprador tanque de aeração intertravado
      "SO-203-06D-YI" : Bool;   // Soprador tanque de aeração intertravado
      "SO-203-06E-YI" : Bool;   // Soprador tanque de aeração intertravado
      "SO-203-06F-YI" : Bool;   // Soprador tanque de aeração intertravado
      "MB-01-YSP" : Bool;   // MB-01 selecionada como principal
      "MB-02-YSP" : Bool;   // MB-02 selecionada como principal
      "MB-04-YSP" : Bool;   // MB-03 selecionada como principal
      "MB-03-YSP" : Bool;   // MB-03 selecionada como principal
      "MB-01-YC1" : Bool;   // MB-01 selecionada como complementar 1
      "MB-02-YC1" : Bool;   // MB-02 selecionada como complementar 1
      "MB-04-YC1" : Bool;   // MB-03 selecionada como complementar 1
      "MB-03-YC1" : Bool;   // MB-03 selecionada como complementar 1
      "MB-01-YC2" : Bool;   // MB-01 selecionada como complementar 2
      "MB-02-YC2" : Bool;   // MB-02 selecionada como complementar 2
      "MB-04-YC2" : Bool;   // MB-03 selecionada como complementar 2
      "MB-03-YC2" : Bool;   // MB-03 selecionada como complementar 2
   END_VAR
BEGIN
END_DATA_BLOCK

DATA_BLOCK "Totalizadores"   // DB306
{ S7_Optimized_Access := 'FALSE' }
VERSION : 0.1
// stored: AutoNumber false, DBAccessibleFromOPCUA true, IsOnlyStoredInLoadMemory false, IsWriteProtectedInAS false
   VAR
      "MB-01-SO" : Int;   // Segundos em operação elevatoria principal
      "MB-01-MO" : Int;   // Minutos em operação elevatoria principal
      "MB-01-HO" : Int;   // Horas em operação elevatoria principal
      "MB-02-SO" : Int;   // Segundos em operação elevatoria principal
      "MB-02-MO" : Int;   // Minutos em operação elevatoria principal
      "MB-02-HO" : Int;   // Horas em operação elevatoria principal
      "MB-03-SO" : Int;   // Segundos em operação elevatoria principal
      "MB-03-MO" : Int;   // Minutos em operação elevatoria principal
      "MB-03-HO" : Int;   // Horas em operação elevatoria principal
      "MB-04-SO" : Int;   // Segundos em operação elevatoria principal
      "MB-04-MO" : Int;   // Minutos em operação elevatoria principal
      "MB-04-HO" : Int;   // Horas em operação elevatoria principal
   END_VAR
BEGIN
END_DATA_BLOCK

DATA_BLOCK "VARIAVEIS"   // DB304
{ S7_Optimized_Access := 'FALSE' }
VERSION : 0.1
// stored: AutoNumber false, DBAccessibleFromOPCUA true, IsOnlyStoredInLoadMemory false, IsWriteProtectedInAS false
   VAR
      "MB-01-YST" : Real;   // Frequência raspador de areia
      "MB-01-YIT" : Real;   // Corrente raspador de areia
      "MB-02-YIT" : Real;   // Corrente raspador de areia
      "MB-02-YST" : Real;   // Frequência raspador de areia
      "MB-03-YIT" : Real;   // Corrente raspador de areia
      "MB-03-YST" : Real;   // Frequência raspador de areia
      "MB-04-YIT" : Real;   // Corrente raspador de areia
      "MB-04-YST" : Real;   // Frequência raspador de areia
      LIT_001 : Real;   // Nível Tanque
      "LIT_001-P" : Real;   // Percentual Tanque
      "PCM-E-CF-01-04-P100-ETRS" : Real;   // Tensão entre fases R e S
      "PCM-E-CF-01-04-P100-ETST" : Real;   // Tensão entre fases S e T
      "PCM-E-CF-01-04-P100-ETTR" : Real;   // Tensão entre fases T e R
      "PCM-E-CF-01-04-P100-ITR" : Real;   // Corrente fase R
      "PCM-E-CF-01-04-P100-ITS" : Real;   // Corrente fase S
      "PCM-E-CF-01-04-P100-ITT" : Real;   // Corrente fase T
      "PCM-E-CF-01-04-P100-JPT" : Real;   // Potência ativa total
      "PCM-E-CF-01-04-P100-JQT" : Real;   // Potência reativa total
      "PCM-E-CF-01-04-P100-JST" : Real;   // Potência aparente total
      "PCM-E-CF-01-04-P100-FP" : Real;   // Fator de potência
      "QGBT-AUX-01-P100-ETRS" : Real;   // Tensão entre fases R e S
      "QGBT-AUX-01-P100-ETST" : Real;   // Tensão entre fases S e T
      "QGBT-AUX-01-P100-ETTR" : Real;   // Tensão entre fases T e R
      "QGBT-AUX-01-P100-ITR" : Real;   // Corrente fase R
      "QGBT-AUX-01-P100-ITS" : Real;   // Corrente fase S
      "QGBT-AUX-01-P100-ITT" : Real;   // Corrente fase T
      "QGBT-AUX-01-P100-JPT" : Real;   // Potência ativa total
      "QGBT-AUX-01-P100-JQT" : Real;   // Potência reativa total
      "QGBT-AUX-01-P100-JST" : Real;   // Potência aparente total
      "QGBT-AUX-01-P100-FP" : Real;   // Fator de potência
   END_VAR
BEGIN
END_DATA_BLOCK

ORGANIZATION_BLOCK "Main"   // OB1, LAD, ProgramCycle
TITLE = "Main Program Sweep (Cycle)"
{ S7_Optimized_Access := 'TRUE' }
VERSION : 0.1
// stored: AutoNumber true, IsIECCheckEnabled false, SetENOAutomatically false
   VAR_INPUT
      Initial_Call : Bool;   // Initial call of this OB
      Remanence : Bool;   // =True, if remanent data are available
   END_VAR
BEGIN

REGION Network 1: PULSO 1 SEGUNDO
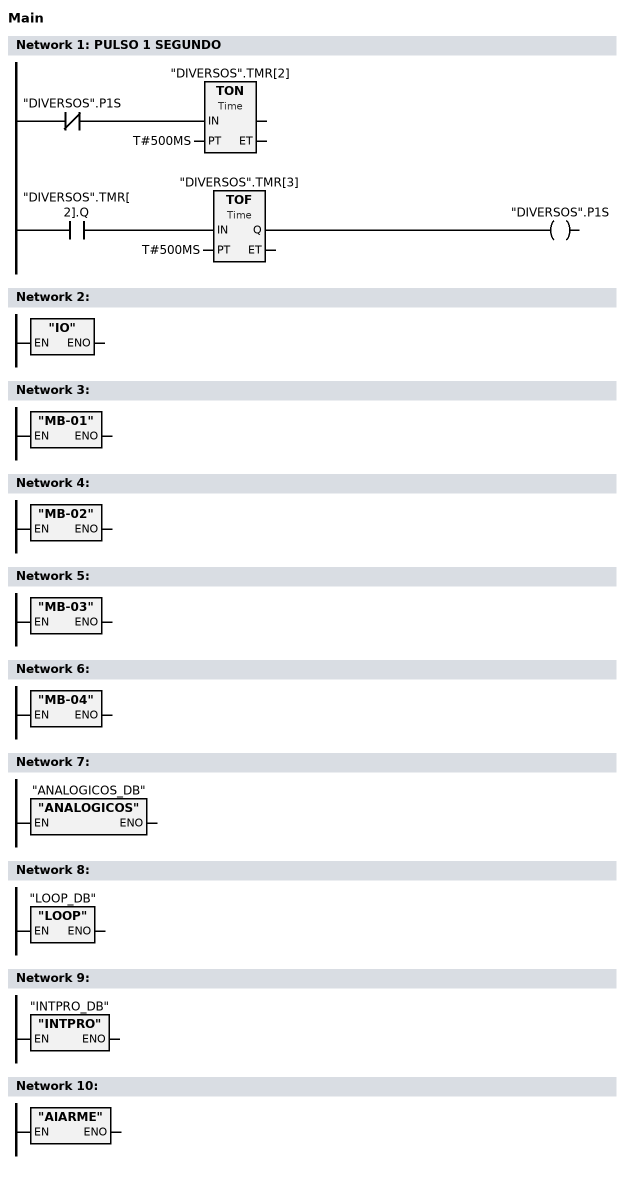
   RUNG wire#powerrail
      I_Contact( "DIVERSOS".P1S )
      { S7_Templates := "time_type := Time" } "DIVERSOS".TMR[2].TON(pt := T#500MS, et =>)
   END_RUNG
   RUNG wire#powerrail
      Contact( "DIVERSOS".TMR[2].Q )
      { S7_Templates := "time_type := Time" } "DIVERSOS".TMR[3].TOF(pt := T#500MS, et =>)
      Coil( "DIVERSOS".P1S )
   END_RUNG
   // the same network as SCL:
   "DIVERSOS".TMR[2].TON(IN := NOT "DIVERSOS".P1S, PT := T#500MS);
   "DIVERSOS".TMR[3].TOF(IN := "DIVERSOS".TMR[2].Q, PT := T#500MS);
   "DIVERSOS".P1S := "DIVERSOS".TMR[3].Q;
END_REGION

REGION Network 2
   RUNG wire#powerrail
      "IO"()
   END_RUNG
   // the same network as SCL:
   "IO"();
END_REGION

REGION Network 3
   RUNG wire#powerrail
      "MB-01"()
   END_RUNG
   // the same network as SCL:
   "MB-01"();
END_REGION

REGION Network 4
   RUNG wire#powerrail
      "MB-02"()
   END_RUNG
   // the same network as SCL:
   "MB-02"();
END_REGION

REGION Network 5
   RUNG wire#powerrail
      "MB-03"()
   END_RUNG
   // the same network as SCL:
   "MB-03"();
END_REGION

REGION Network 6
   RUNG wire#powerrail
      "MB-04"()
   END_RUNG
   // the same network as SCL:
   "MB-04"();
END_REGION

REGION Network 7
   RUNG wire#powerrail
      "ANALOGICOS_DB"()
   END_RUNG
   // the same network as SCL:
   "ANALOGICOS_DB"();   // "ANALOGICOS"
END_REGION

REGION Network 8
   RUNG wire#powerrail
      "LOOP_DB"()
   END_RUNG
   // the same network as SCL:
   "LOOP_DB"();   // "LOOP"
END_REGION

REGION Network 9
   RUNG wire#powerrail
      "INTPRO_DB"()
   END_RUNG
   // the same network as SCL:
   "INTPRO_DB"();   // "INTPRO"
END_REGION

REGION Network 10
   RUNG wire#powerrail
      "AlARME"()
   END_RUNG
   // the same network as SCL:
   "AlARME"();
END_REGION
END_ORGANIZATION_BLOCK

FUNCTION "IO" : Void   // FC1, LAD
{ S7_Optimized_Access := 'TRUE' }
VERSION : 0.1
// stored: AutoNumber false, IsIECCheckEnabled false, SetENOAutomatically false, UDAEnableTagReadback false
BEGIN

REGION Network 1: Status e alarme elevatória principal 1
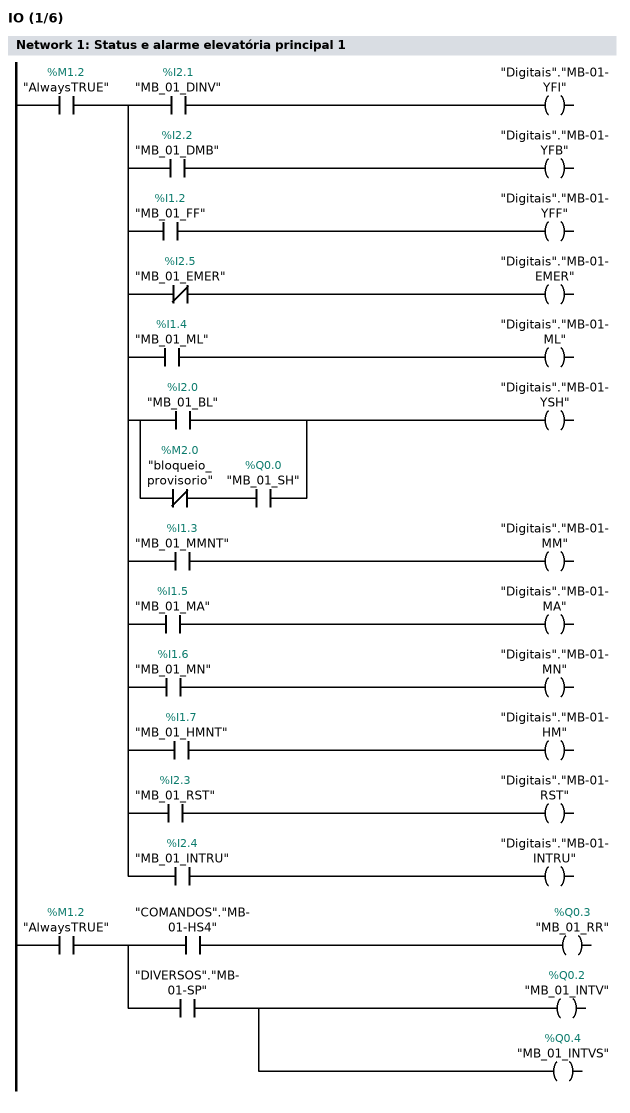
   RUNG wire#powerrail
      Contact( "AlwaysTRUE" )
      wire#w1
      Contact( "MB_01_DINV" )
      Coil( "Digitais"."MB-01-YFI" )
   END_RUNG
   RUNG wire#w1
      Contact( "MB_01_DMB" )
      Coil( "Digitais"."MB-01-YFB" )
   END_RUNG
   RUNG wire#w1
      Contact( "MB_01_FF" )
      Coil( "Digitais"."MB-01-YFF" )
   END_RUNG
   RUNG wire#w1
      I_Contact( "MB_01_EMER" )
      Coil( "Digitais"."MB-01-EMER" )
   END_RUNG
   RUNG wire#w1
      Contact( "MB_01_ML" )
      Coil( "Digitais"."MB-01-ML" )
   END_RUNG
   RUNG wire#w1
      Contact( "MB_01_BL" )
      wire#w2
      Coil( "Digitais"."MB-01-YSH" )
   END_RUNG
   RUNG wire#w1
      I_Contact( "bloqueio_provisorio" )
      Contact( "MB_01_SH" )
   END_RUNG wire#w2
   RUNG wire#w1
      Contact( "MB_01_MMNT" )
      Coil( "Digitais"."MB-01-MM" )
   END_RUNG
   RUNG wire#w1
      Contact( "MB_01_MA" )
      Coil( "Digitais"."MB-01-MA" )
   END_RUNG
   RUNG wire#w1
      Contact( "MB_01_MN" )
      Coil( "Digitais"."MB-01-MN" )
   END_RUNG
   RUNG wire#w1
      Contact( "MB_01_HMNT" )
      Coil( "Digitais"."MB-01-HM" )
   END_RUNG
   RUNG wire#w1
      Contact( "MB_01_RST" )
      Coil( "Digitais"."MB-01-RST" )
   END_RUNG
   RUNG wire#w1
      Contact( "MB_01_INTRU" )
      Coil( "Digitais"."MB-01-INTRU" )
   END_RUNG
   RUNG wire#powerrail
      Contact( "AlwaysTRUE" )
      wire#w3
      Contact( "COMANDOS"."MB-01-HS4" )
      Coil( "MB_01_RR" )
   END_RUNG
   RUNG wire#w3
      Contact( "DIVERSOS"."MB-01-SP" )
      wire#w4
      Coil( "MB_01_INTV" )
   END_RUNG
   RUNG wire#w4
      Coil( "MB_01_INTVS" )
   END_RUNG
   // the same network as SCL:
   "Digitais"."MB-01-YFI" := "AlwaysTRUE" AND "MB_01_DINV";
   "Digitais"."MB-01-YFB" := "AlwaysTRUE" AND "MB_01_DMB";
   "Digitais"."MB-01-YFF" := "AlwaysTRUE" AND "MB_01_FF";
   "Digitais"."MB-01-EMER" := "AlwaysTRUE" AND NOT "MB_01_EMER";
   "Digitais"."MB-01-ML" := "AlwaysTRUE" AND "MB_01_ML";
   "Digitais"."MB-01-YSH" := "AlwaysTRUE" AND ("MB_01_BL" OR (NOT "bloqueio_provisorio" AND "MB_01_SH"));
   "Digitais"."MB-01-MM" := "AlwaysTRUE" AND "MB_01_MMNT";
   "Digitais"."MB-01-MA" := "AlwaysTRUE" AND "MB_01_MA";
   "Digitais"."MB-01-MN" := "AlwaysTRUE" AND "MB_01_MN";
   "Digitais"."MB-01-HM" := "AlwaysTRUE" AND "MB_01_HMNT";
   "Digitais"."MB-01-RST" := "AlwaysTRUE" AND "MB_01_RST";
   "Digitais"."MB-01-INTRU" := "AlwaysTRUE" AND "MB_01_INTRU";
   "MB_01_RR" := "AlwaysTRUE" AND "COMANDOS"."MB-01-HS4";
   "MB_01_INTV" := "AlwaysTRUE" AND "DIVERSOS"."MB-01-SP";
   "MB_01_INTVS" := "MB_01_INTV";
END_REGION

REGION Network 2: Status e alarme elevatória principal 2
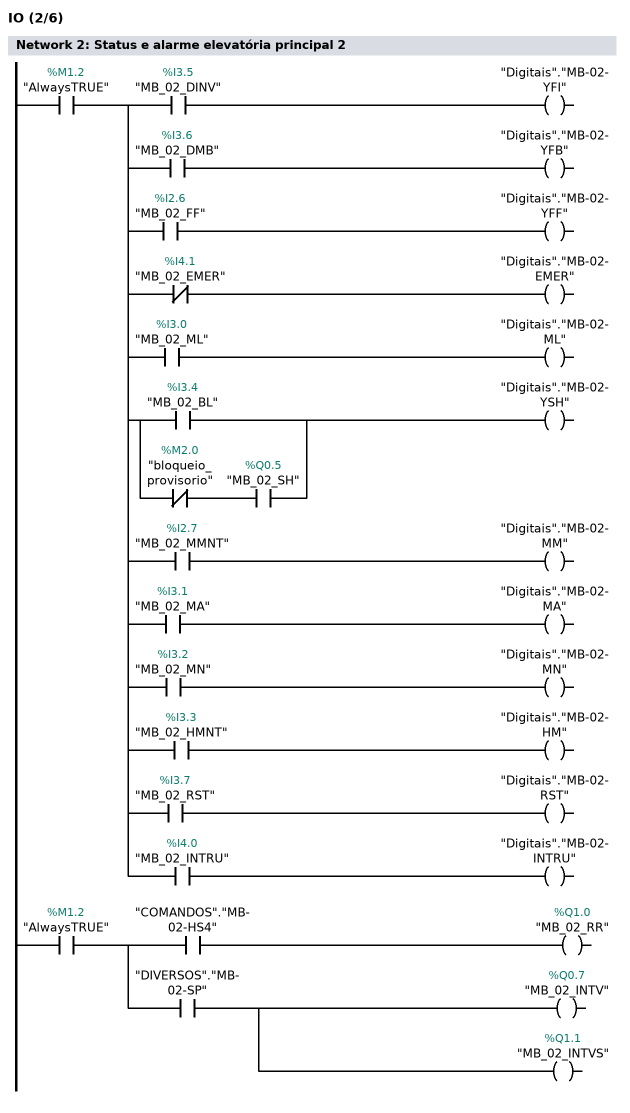
   RUNG wire#powerrail
      Contact( "AlwaysTRUE" )
      wire#w1
      Contact( "MB_02_DINV" )
      Coil( "Digitais"."MB-02-YFI" )
   END_RUNG
   RUNG wire#w1
      Contact( "MB_02_DMB" )
      Coil( "Digitais"."MB-02-YFB" )
   END_RUNG
   RUNG wire#w1
      Contact( "MB_02_FF" )
      Coil( "Digitais"."MB-02-YFF" )
   END_RUNG
   RUNG wire#w1
      I_Contact( "MB_02_EMER" )
      Coil( "Digitais"."MB-02-EMER" )
   END_RUNG
   RUNG wire#w1
      Contact( "MB_02_ML" )
      Coil( "Digitais"."MB-02-ML" )
   END_RUNG
   RUNG wire#w1
      Contact( "MB_02_BL" )
      wire#w2
      Coil( "Digitais"."MB-02-YSH" )
   END_RUNG
   RUNG wire#w1
      I_Contact( "bloqueio_provisorio" )
      Contact( "MB_02_SH" )
   END_RUNG wire#w2
   RUNG wire#w1
      Contact( "MB_02_MMNT" )
      Coil( "Digitais"."MB-02-MM" )
   END_RUNG
   RUNG wire#w1
      Contact( "MB_02_MA" )
      Coil( "Digitais"."MB-02-MA" )
   END_RUNG
   RUNG wire#w1
      Contact( "MB_02_MN" )
      Coil( "Digitais"."MB-02-MN" )
   END_RUNG
   RUNG wire#w1
      Contact( "MB_02_HMNT" )
      Coil( "Digitais"."MB-02-HM" )
   END_RUNG
   RUNG wire#w1
      Contact( "MB_02_RST" )
      Coil( "Digitais"."MB-02-RST" )
   END_RUNG
   RUNG wire#w1
      Contact( "MB_02_INTRU" )
      Coil( "Digitais"."MB-02-INTRU" )
   END_RUNG
   RUNG wire#powerrail
      Contact( "AlwaysTRUE" )
      wire#w3
      Contact( "COMANDOS"."MB-02-HS4" )
      Coil( "MB_02_RR" )
   END_RUNG
   RUNG wire#w3
      Contact( "DIVERSOS"."MB-02-SP" )
      wire#w4
      Coil( "MB_02_INTV" )
   END_RUNG
   RUNG wire#w4
      Coil( "MB_02_INTVS" )
   END_RUNG
   // the same network as SCL:
   "Digitais"."MB-02-YFI" := "AlwaysTRUE" AND "MB_02_DINV";
   "Digitais"."MB-02-YFB" := "AlwaysTRUE" AND "MB_02_DMB";
   "Digitais"."MB-02-YFF" := "AlwaysTRUE" AND "MB_02_FF";
   "Digitais"."MB-02-EMER" := "AlwaysTRUE" AND NOT "MB_02_EMER";
   "Digitais"."MB-02-ML" := "AlwaysTRUE" AND "MB_02_ML";
   "Digitais"."MB-02-YSH" := "AlwaysTRUE" AND ("MB_02_BL" OR (NOT "bloqueio_provisorio" AND "MB_02_SH"));
   "Digitais"."MB-02-MM" := "AlwaysTRUE" AND "MB_02_MMNT";
   "Digitais"."MB-02-MA" := "AlwaysTRUE" AND "MB_02_MA";
   "Digitais"."MB-02-MN" := "AlwaysTRUE" AND "MB_02_MN";
   "Digitais"."MB-02-HM" := "AlwaysTRUE" AND "MB_02_HMNT";
   "Digitais"."MB-02-RST" := "AlwaysTRUE" AND "MB_02_RST";
   "Digitais"."MB-02-INTRU" := "AlwaysTRUE" AND "MB_02_INTRU";
   "MB_02_RR" := "AlwaysTRUE" AND "COMANDOS"."MB-02-HS4";
   "MB_02_INTV" := "AlwaysTRUE" AND "DIVERSOS"."MB-02-SP";
   "MB_02_INTVS" := "MB_02_INTV";
END_REGION

REGION Network 3: Status e alarme elevatória principal 3
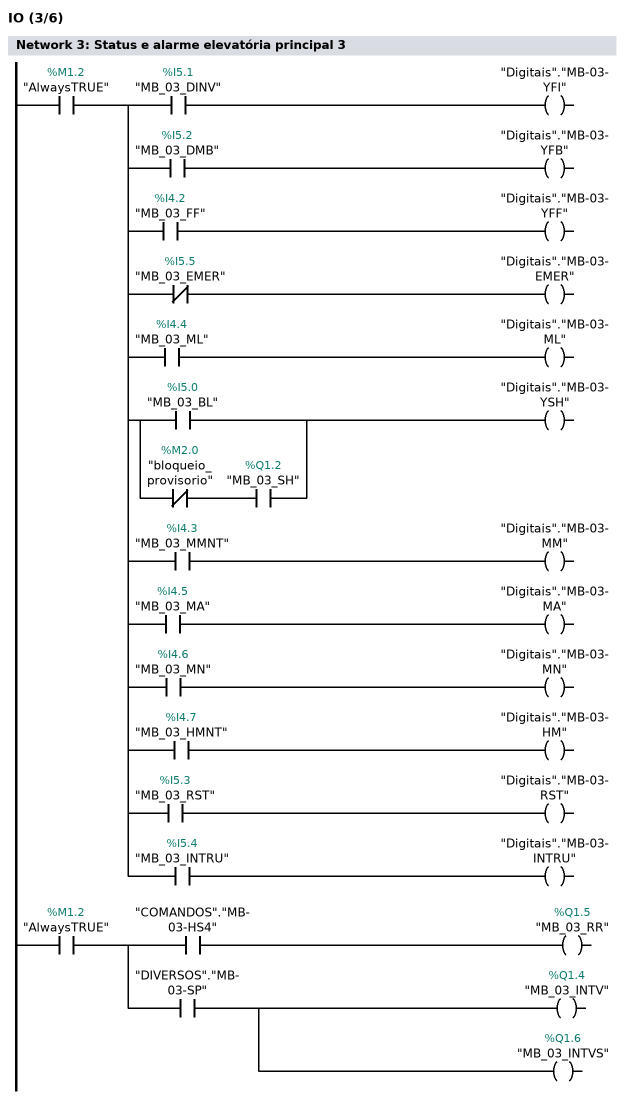
   RUNG wire#powerrail
      Contact( "AlwaysTRUE" )
      wire#w1
      Contact( "MB_03_DINV" )
      Coil( "Digitais"."MB-03-YFI" )
   END_RUNG
   RUNG wire#w1
      Contact( "MB_03_DMB" )
      Coil( "Digitais"."MB-03-YFB" )
   END_RUNG
   RUNG wire#w1
      Contact( "MB_03_FF" )
      Coil( "Digitais"."MB-03-YFF" )
   END_RUNG
   RUNG wire#w1
      I_Contact( "MB_03_EMER" )
      Coil( "Digitais"."MB-03-EMER" )
   END_RUNG
   RUNG wire#w1
      Contact( "MB_03_ML" )
      Coil( "Digitais"."MB-03-ML" )
   END_RUNG
   RUNG wire#w1
      Contact( "MB_03_BL" )
      wire#w2
      Coil( "Digitais"."MB-03-YSH" )
   END_RUNG
   RUNG wire#w1
      I_Contact( "bloqueio_provisorio" )
      Contact( "MB_03_SH" )
   END_RUNG wire#w2
   RUNG wire#w1
      Contact( "MB_03_MMNT" )
      Coil( "Digitais"."MB-03-MM" )
   END_RUNG
   RUNG wire#w1
      Contact( "MB_03_MA" )
      Coil( "Digitais"."MB-03-MA" )
   END_RUNG
   RUNG wire#w1
      Contact( "MB_03_MN" )
      Coil( "Digitais"."MB-03-MN" )
   END_RUNG
   RUNG wire#w1
      Contact( "MB_03_HMNT" )
      Coil( "Digitais"."MB-03-HM" )
   END_RUNG
   RUNG wire#w1
      Contact( "MB_03_RST" )
      Coil( "Digitais"."MB-03-RST" )
   END_RUNG
   RUNG wire#w1
      Contact( "MB_03_INTRU" )
      Coil( "Digitais"."MB-03-INTRU" )
   END_RUNG
   RUNG wire#powerrail
      Contact( "AlwaysTRUE" )
      wire#w3
      Contact( "COMANDOS"."MB-03-HS4" )
      Coil( "MB_03_RR" )
   END_RUNG
   RUNG wire#w3
      Contact( "DIVERSOS"."MB-03-SP" )
      wire#w4
      Coil( "MB_03_INTV" )
   END_RUNG
   RUNG wire#w4
      Coil( "MB_03_INTVS" )
   END_RUNG
   // the same network as SCL:
   "Digitais"."MB-03-YFI" := "AlwaysTRUE" AND "MB_03_DINV";
   "Digitais"."MB-03-YFB" := "AlwaysTRUE" AND "MB_03_DMB";
   "Digitais"."MB-03-YFF" := "AlwaysTRUE" AND "MB_03_FF";
   "Digitais"."MB-03-EMER" := "AlwaysTRUE" AND NOT "MB_03_EMER";
   "Digitais"."MB-03-ML" := "AlwaysTRUE" AND "MB_03_ML";
   "Digitais"."MB-03-YSH" := "AlwaysTRUE" AND ("MB_03_BL" OR (NOT "bloqueio_provisorio" AND "MB_03_SH"));
   "Digitais"."MB-03-MM" := "AlwaysTRUE" AND "MB_03_MMNT";
   "Digitais"."MB-03-MA" := "AlwaysTRUE" AND "MB_03_MA";
   "Digitais"."MB-03-MN" := "AlwaysTRUE" AND "MB_03_MN";
   "Digitais"."MB-03-HM" := "AlwaysTRUE" AND "MB_03_HMNT";
   "Digitais"."MB-03-RST" := "AlwaysTRUE" AND "MB_03_RST";
   "Digitais"."MB-03-INTRU" := "AlwaysTRUE" AND "MB_03_INTRU";
   "MB_03_RR" := "AlwaysTRUE" AND "COMANDOS"."MB-03-HS4";
   "MB_03_INTV" := "AlwaysTRUE" AND "DIVERSOS"."MB-03-SP";
   "MB_03_INTVS" := "MB_03_INTV";
END_REGION

REGION Network 4: Status e alarme elevatória principal 4
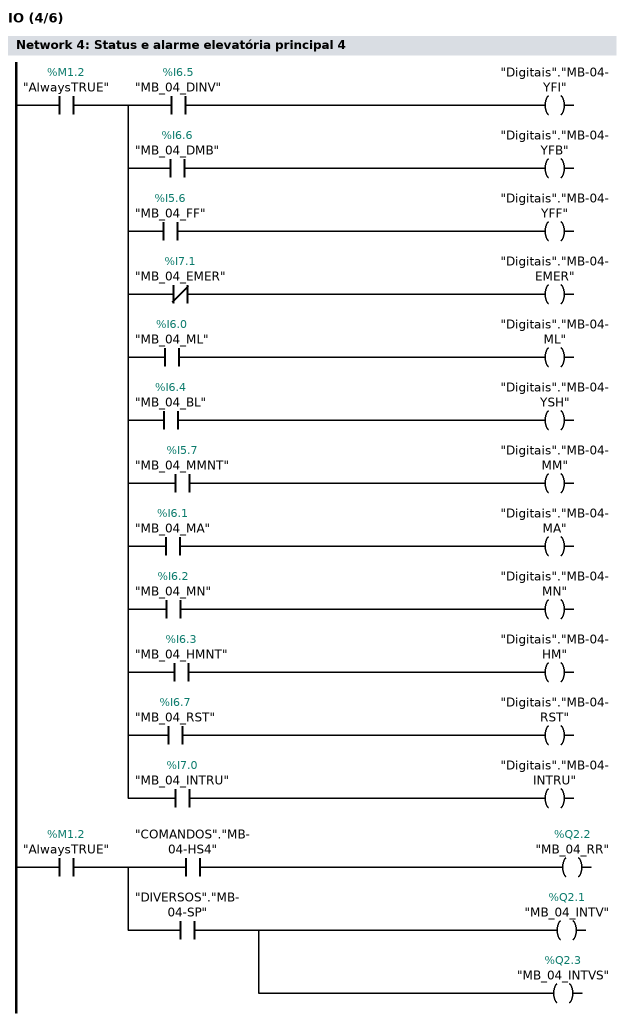
   RUNG wire#powerrail
      Contact( "AlwaysTRUE" )
      wire#w1
      Contact( "MB_04_DINV" )
      Coil( "Digitais"."MB-04-YFI" )
   END_RUNG
   RUNG wire#w1
      Contact( "MB_04_DMB" )
      Coil( "Digitais"."MB-04-YFB" )
   END_RUNG
   RUNG wire#w1
      Contact( "MB_04_FF" )
      Coil( "Digitais"."MB-04-YFF" )
   END_RUNG
   RUNG wire#w1
      I_Contact( "MB_04_EMER" )
      Coil( "Digitais"."MB-04-EMER" )
   END_RUNG
   RUNG wire#w1
      Contact( "MB_04_ML" )
      Coil( "Digitais"."MB-04-ML" )
   END_RUNG
   RUNG wire#w1
      Contact( "MB_04_BL" )
      Coil( "Digitais"."MB-04-YSH" )
   END_RUNG
   RUNG wire#w1
      Contact( "MB_04_MMNT" )
      Coil( "Digitais"."MB-04-MM" )
   END_RUNG
   RUNG wire#w1
      Contact( "MB_04_MA" )
      Coil( "Digitais"."MB-04-MA" )
   END_RUNG
   RUNG wire#w1
      Contact( "MB_04_MN" )
      Coil( "Digitais"."MB-04-MN" )
   END_RUNG
   RUNG wire#w1
      Contact( "MB_04_HMNT" )
      Coil( "Digitais"."MB-04-HM" )
   END_RUNG
   RUNG wire#w1
      Contact( "MB_04_RST" )
      Coil( "Digitais"."MB-04-RST" )
   END_RUNG
   RUNG wire#w1
      Contact( "MB_04_INTRU" )
      Coil( "Digitais"."MB-04-INTRU" )
   END_RUNG
   RUNG wire#powerrail
      Contact( "AlwaysTRUE" )
      wire#w2
      Contact( "COMANDOS"."MB-04-HS4" )
      Coil( "MB_04_RR" )
   END_RUNG
   RUNG wire#w2
      Contact( "DIVERSOS"."MB-04-SP" )
      wire#w3
      Coil( "MB_04_INTV" )
   END_RUNG
   RUNG wire#w3
      Coil( "MB_04_INTVS" )
   END_RUNG
   // the same network as SCL:
   "Digitais"."MB-04-YFI" := "AlwaysTRUE" AND "MB_04_DINV";
   "Digitais"."MB-04-YFB" := "AlwaysTRUE" AND "MB_04_DMB";
   "Digitais"."MB-04-YFF" := "AlwaysTRUE" AND "MB_04_FF";
   "Digitais"."MB-04-EMER" := "AlwaysTRUE" AND NOT "MB_04_EMER";
   "Digitais"."MB-04-ML" := "AlwaysTRUE" AND "MB_04_ML";
   "Digitais"."MB-04-YSH" := "AlwaysTRUE" AND "MB_04_BL";
   "Digitais"."MB-04-MM" := "AlwaysTRUE" AND "MB_04_MMNT";
   "Digitais"."MB-04-MA" := "AlwaysTRUE" AND "MB_04_MA";
   "Digitais"."MB-04-MN" := "AlwaysTRUE" AND "MB_04_MN";
   "Digitais"."MB-04-HM" := "AlwaysTRUE" AND "MB_04_HMNT";
   "Digitais"."MB-04-RST" := "AlwaysTRUE" AND "MB_04_RST";
   "Digitais"."MB-04-INTRU" := "AlwaysTRUE" AND "MB_04_INTRU";
   "MB_04_RR" := "AlwaysTRUE" AND "COMANDOS"."MB-04-HS4";
   "MB_04_INTV" := "AlwaysTRUE" AND "DIVERSOS"."MB-04-SP";
   "MB_04_INTVS" := "MB_04_INTV";
END_REGION

REGION Network 5: Status e alarme PCM-E-CF-01-04
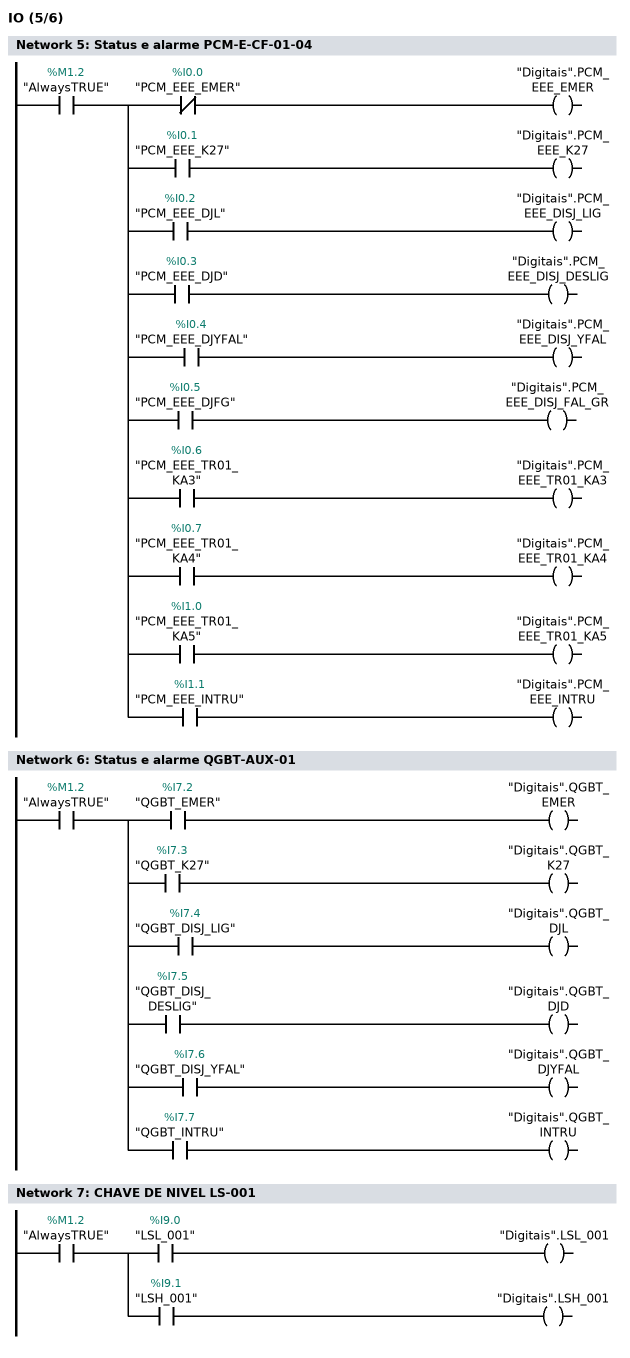
   RUNG wire#powerrail
      Contact( "AlwaysTRUE" )
      wire#w1
      I_Contact( "PCM_EEE_EMER" )
      Coil( "Digitais".PCM_EEE_EMER )
   END_RUNG
   RUNG wire#w1
      Contact( "PCM_EEE_K27" )
      Coil( "Digitais".PCM_EEE_K27 )
   END_RUNG
   RUNG wire#w1
      Contact( "PCM_EEE_DJL" )
      Coil( "Digitais".PCM_EEE_DISJ_LIG )
   END_RUNG
   RUNG wire#w1
      Contact( "PCM_EEE_DJD" )
      Coil( "Digitais".PCM_EEE_DISJ_DESLIG )
   END_RUNG
   RUNG wire#w1
      Contact( "PCM_EEE_DJYFAL" )
      Coil( "Digitais".PCM_EEE_DISJ_YFAL )
   END_RUNG
   RUNG wire#w1
      Contact( "PCM_EEE_DJFG" )
      Coil( "Digitais".PCM_EEE_DISJ_FAL_GR )
   END_RUNG
   RUNG wire#w1
      Contact( "PCM_EEE_TR01_KA3" )
      Coil( "Digitais".PCM_EEE_TR01_KA3 )
   END_RUNG
   RUNG wire#w1
      Contact( "PCM_EEE_TR01_KA4" )
      Coil( "Digitais".PCM_EEE_TR01_KA4 )
   END_RUNG
   RUNG wire#w1
      Contact( "PCM_EEE_TR01_KA5" )
      Coil( "Digitais".PCM_EEE_TR01_KA5 )
   END_RUNG
   RUNG wire#w1
      Contact( "PCM_EEE_INTRU" )
      Coil( "Digitais".PCM_EEE_INTRU )
   END_RUNG
   // the same network as SCL:
   "Digitais".PCM_EEE_EMER := "AlwaysTRUE" AND NOT "PCM_EEE_EMER";
   "Digitais".PCM_EEE_K27 := "AlwaysTRUE" AND "PCM_EEE_K27";
   "Digitais".PCM_EEE_DISJ_LIG := "AlwaysTRUE" AND "PCM_EEE_DJL";
   "Digitais".PCM_EEE_DISJ_DESLIG := "AlwaysTRUE" AND "PCM_EEE_DJD";
   "Digitais".PCM_EEE_DISJ_YFAL := "AlwaysTRUE" AND "PCM_EEE_DJYFAL";
   "Digitais".PCM_EEE_DISJ_FAL_GR := "AlwaysTRUE" AND "PCM_EEE_DJFG";
   "Digitais".PCM_EEE_TR01_KA3 := "AlwaysTRUE" AND "PCM_EEE_TR01_KA3";
   "Digitais".PCM_EEE_TR01_KA4 := "AlwaysTRUE" AND "PCM_EEE_TR01_KA4";
   "Digitais".PCM_EEE_TR01_KA5 := "AlwaysTRUE" AND "PCM_EEE_TR01_KA5";
   "Digitais".PCM_EEE_INTRU := "AlwaysTRUE" AND "PCM_EEE_INTRU";
END_REGION

REGION Network 6: Status e alarme QGBT-AUX-01
   RUNG wire#powerrail
      Contact( "AlwaysTRUE" )
      wire#w1
      Contact( "QGBT_EMER" )
      Coil( "Digitais".QGBT_EMER )
   END_RUNG
   RUNG wire#w1
      Contact( "QGBT_K27" )
      Coil( "Digitais".QGBT_K27 )
   END_RUNG
   RUNG wire#w1
      Contact( "QGBT_DISJ_LIG" )
      Coil( "Digitais".QGBT_DJL )
   END_RUNG
   RUNG wire#w1
      Contact( "QGBT_DISJ_DESLIG" )
      Coil( "Digitais".QGBT_DJD )
   END_RUNG
   RUNG wire#w1
      Contact( "QGBT_DISJ_YFAL" )
      Coil( "Digitais".QGBT_DJYFAL )
   END_RUNG
   RUNG wire#w1
      Contact( "QGBT_INTRU" )
      Coil( "Digitais".QGBT_INTRU )
   END_RUNG
   // the same network as SCL:
   "Digitais".QGBT_EMER := "AlwaysTRUE" AND "QGBT_EMER";
   "Digitais".QGBT_K27 := "AlwaysTRUE" AND "QGBT_K27";
   "Digitais".QGBT_DJL := "AlwaysTRUE" AND "QGBT_DISJ_LIG";
   "Digitais".QGBT_DJD := "AlwaysTRUE" AND "QGBT_DISJ_DESLIG";
   "Digitais".QGBT_DJYFAL := "AlwaysTRUE" AND "QGBT_DISJ_YFAL";
   "Digitais".QGBT_INTRU := "AlwaysTRUE" AND "QGBT_INTRU";
END_REGION

REGION Network 7: CHAVE DE NIVEL LS-001
   RUNG wire#powerrail
      Contact( "AlwaysTRUE" )
      wire#w1
      Contact( "LSL_001" )
      Coil( "Digitais".LSL_001 )
   END_RUNG
   RUNG wire#w1
      Contact( "LSH_001" )
      Coil( "Digitais".LSH_001 )
   END_RUNG
   // the same network as SCL:
   "Digitais".LSL_001 := "AlwaysTRUE" AND "LSL_001";
   "Digitais".LSH_001 := "AlwaysTRUE" AND "LSH_001";
END_REGION

REGION Network 8: CHAVE DE NIVEL LS-002
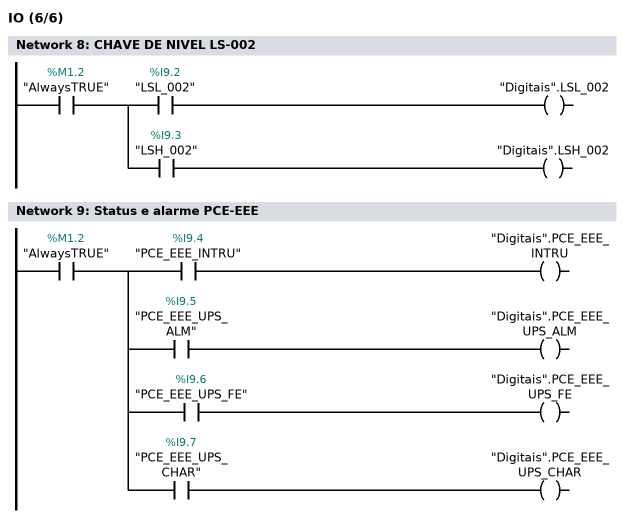
   RUNG wire#powerrail
      Contact( "AlwaysTRUE" )
      wire#w1
      Contact( "LSL_002" )
      Coil( "Digitais".LSL_002 )
   END_RUNG
   RUNG wire#w1
      Contact( "LSH_002" )
      Coil( "Digitais".LSH_002 )
   END_RUNG
   // the same network as SCL:
   "Digitais".LSL_002 := "AlwaysTRUE" AND "LSL_002";
   "Digitais".LSH_002 := "AlwaysTRUE" AND "LSH_002";
END_REGION

REGION Network 9: Status e alarme PCE-EEE
   RUNG wire#powerrail
      Contact( "AlwaysTRUE" )
      wire#w1
      Contact( "PCE_EEE_INTRU" )
      Coil( "Digitais".PCE_EEE_INTRU )
   END_RUNG
   RUNG wire#w1
      Contact( "PCE_EEE_UPS_ALM" )
      Coil( "Digitais".PCE_EEE_UPS_ALM )
   END_RUNG
   RUNG wire#w1
      Contact( "PCE_EEE_UPS_FE" )
      Coil( "Digitais".PCE_EEE_UPS_FE )
   END_RUNG
   RUNG wire#w1
      Contact( "PCE_EEE_UPS_CHAR" )
      Coil( "Digitais".PCE_EEE_UPS_CHAR )
   END_RUNG
   // the same network as SCL:
   "Digitais".PCE_EEE_INTRU := "AlwaysTRUE" AND "PCE_EEE_INTRU";
   "Digitais".PCE_EEE_UPS_ALM := "AlwaysTRUE" AND "PCE_EEE_UPS_ALM";
   "Digitais".PCE_EEE_UPS_FE := "AlwaysTRUE" AND "PCE_EEE_UPS_FE";
   "Digitais".PCE_EEE_UPS_CHAR := "AlwaysTRUE" AND "PCE_EEE_UPS_CHAR";
END_REGION
END_FUNCTION

FUNCTION "MB-01" : Void   // FC22, LAD
TITLE = Lógica de acionamento do motor
{ S7_Optimized_Access := 'FALSE' }
VERSION : 0.1
// stored: AutoNumber false, IsIECCheckEnabled false, SetENOAutomatically false, UDAEnableTagReadback false
   VAR_TEMP
      IM : Bool;   // Intertravamento manual = 0
      IA : Bool;   // Intertravamento automáticol = 0
      HABM : Bool;   // Habilita funcionamento manual = 1
      HABA : Bool;   // Habilita funcionamento automático = 1
      CLM : Bool;   // Comando liga motor
      PROT : Bool;   // Proteção do motor acionada
   END_VAR
BEGIN

REGION Network 1: Intertravamento maual/automático
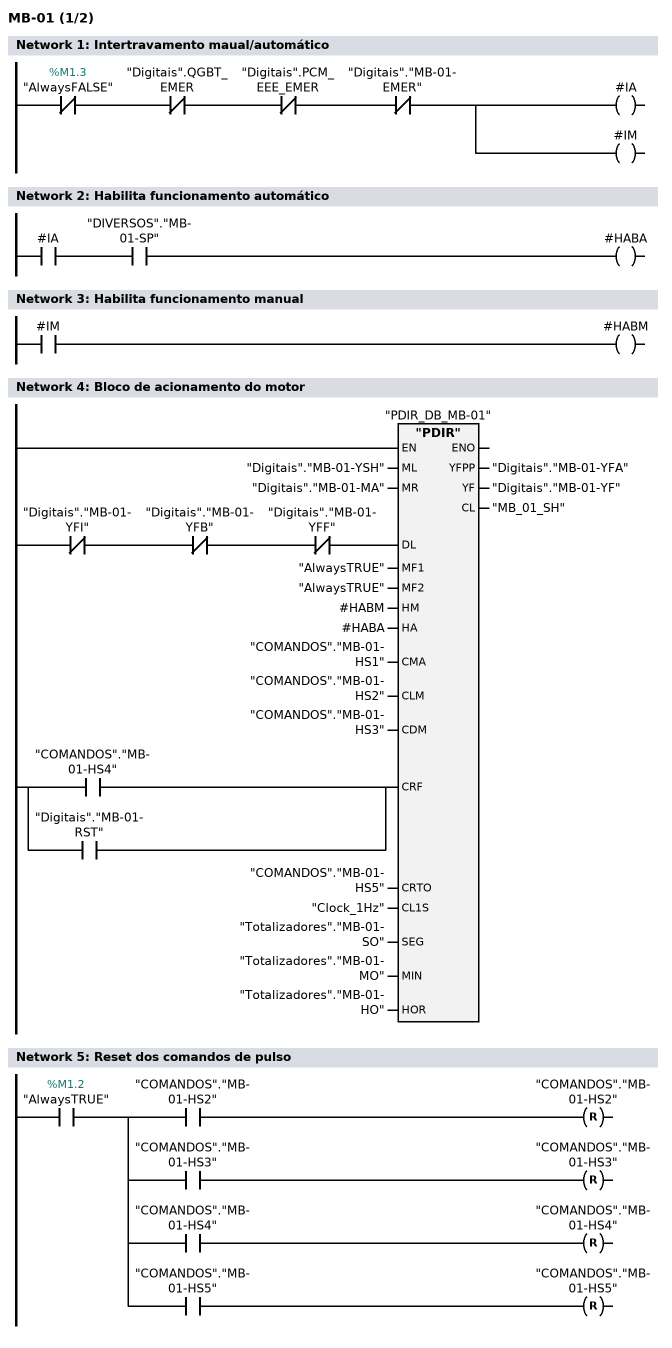
   RUNG wire#powerrail
      I_Contact( "AlwaysFALSE" )
      I_Contact( "Digitais".QGBT_EMER )
      I_Contact( "Digitais".PCM_EEE_EMER )
      I_Contact( "Digitais"."MB-01-EMER" )
      wire#w1
      Coil( #IA )
   END_RUNG
   RUNG wire#w1
      Coil( #IM )
   END_RUNG
   // the same network as SCL:
   #IA := NOT "AlwaysFALSE" AND NOT "Digitais".QGBT_EMER AND NOT "Digitais".PCM_EEE_EMER AND NOT "Digitais"."MB-01-EMER";
   #IM := #IA;
END_REGION

REGION Network 2: Habilita funcionamento automático
   RUNG wire#powerrail
      Contact( #IA )
      Contact( "DIVERSOS"."MB-01-SP" )
      Coil( #HABA )
   END_RUNG
   // the same network as SCL:
   #HABA := #IA AND "DIVERSOS"."MB-01-SP";
END_REGION

REGION Network 3: Habilita funcionamento manual
   RUNG wire#powerrail
      Contact( #IM )
      Coil( #HABM )
   END_RUNG
   // the same network as SCL:
   #HABM := #IM;
END_REGION

REGION Network 4: Bloco de acionamento do motor
   RUNG wire#powerrail
      "PDIR_DB_MB-01"(DL := wire#w1, CRF := wire#w2, ML := "Digitais"."MB-01-YSH", MR := "Digitais"."MB-01-MA", MF1 := "AlwaysTRUE", MF2 := "AlwaysTRUE", HM := #HABM, HA := #HABA, CMA := "COMANDOS"."MB-01-HS1", CLM := "COMANDOS"."MB-01-HS2", CDM := "COMANDOS"."MB-01-HS3", CRTO := "COMANDOS"."MB-01-HS5", CL1S := "Clock_1Hz", SEG := "Totalizadores"."MB-01-SO", MIN := "Totalizadores"."MB-01-MO", HOR := "Totalizadores"."MB-01-HO", YFPP => "Digitais"."MB-01-YFA", YF => "Digitais"."MB-01-YF", CL => "MB_01_SH")
   END_RUNG
   RUNG wire#powerrail
      I_Contact( "Digitais"."MB-01-YFI" )
      I_Contact( "Digitais"."MB-01-YFB" )
      I_Contact( "Digitais"."MB-01-YFF" )
   END_RUNG wire#w1
   RUNG wire#powerrail
      Contact( "COMANDOS"."MB-01-HS4" )
   END_RUNG wire#w2
   RUNG wire#powerrail
      Contact( "Digitais"."MB-01-RST" )
   END_RUNG wire#w2
   // the same network as SCL:
   "PDIR_DB_MB-01"(ML := "Digitais"."MB-01-YSH",   // "PDIR"
                   MR := "Digitais"."MB-01-MA",
                   DL := NOT "Digitais"."MB-01-YFI" AND NOT "Digitais"."MB-01-YFB" AND NOT "Digitais"."MB-01-YFF",
                   MF1 := "AlwaysTRUE",
                   MF2 := "AlwaysTRUE",
                   HM := #HABM,
                   HA := #HABA,
                   CMA := "COMANDOS"."MB-01-HS1",
                   CLM := "COMANDOS"."MB-01-HS2",
                   CDM := "COMANDOS"."MB-01-HS3",
                   CRF := "COMANDOS"."MB-01-HS4" OR "Digitais"."MB-01-RST",
                   CRTO := "COMANDOS"."MB-01-HS5",
                   CL1S := "Clock_1Hz",
                   SEG := "Totalizadores"."MB-01-SO",
                   MIN := "Totalizadores"."MB-01-MO",
                   HOR := "Totalizadores"."MB-01-HO",
                   YFPP => "Digitais"."MB-01-YFA",
                   YF => "Digitais"."MB-01-YF",
                   CL => "MB_01_SH");
END_REGION

REGION Network 5: Reset dos comandos de pulso
   RUNG wire#powerrail
      Contact( "AlwaysTRUE" )
      wire#w1
      Contact( "COMANDOS"."MB-01-HS2" )
      R_Coil( "COMANDOS"."MB-01-HS2" )
   END_RUNG
   RUNG wire#w1
      Contact( "COMANDOS"."MB-01-HS3" )
      R_Coil( "COMANDOS"."MB-01-HS3" )
   END_RUNG
   RUNG wire#w1
      Contact( "COMANDOS"."MB-01-HS4" )
      R_Coil( "COMANDOS"."MB-01-HS4" )
   END_RUNG
   RUNG wire#w1
      Contact( "COMANDOS"."MB-01-HS5" )
      R_Coil( "COMANDOS"."MB-01-HS5" )
   END_RUNG
   // the same network as SCL:
   IF "AlwaysTRUE" AND "COMANDOS"."MB-01-HS2" THEN "COMANDOS"."MB-01-HS2" := FALSE; END_IF;
   IF "AlwaysTRUE" AND "COMANDOS"."MB-01-HS3" THEN "COMANDOS"."MB-01-HS3" := FALSE; END_IF;
   IF "AlwaysTRUE" AND "COMANDOS"."MB-01-HS4" THEN "COMANDOS"."MB-01-HS4" := FALSE; END_IF;
   IF "AlwaysTRUE" AND "COMANDOS"."MB-01-HS5" THEN "COMANDOS"."MB-01-HS5" := FALSE; END_IF;
END_REGION

REGION Network 6: Elevatoria principal modo automatico
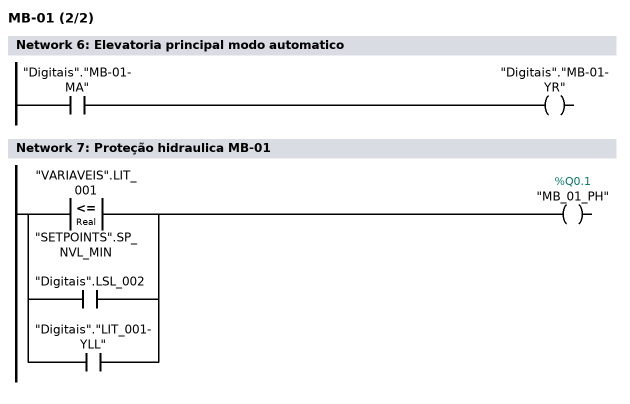
   RUNG wire#powerrail
      Contact( "Digitais"."MB-01-MA" )
      Coil( "Digitais"."MB-01-YR" )
   END_RUNG
   // the same network as SCL:
   "Digitais"."MB-01-YR" := "Digitais"."MB-01-MA";
END_REGION

REGION Network 7: Proteção hidraulica MB-01
   RUNG wire#powerrail
      { S7_Templates := "SrcType := Real" } LE_Contact(in1 := "VARIAVEIS".LIT_001, in2 := "SETPOINTS".SP_NVL_MIN)
      wire#w1
      Coil( "MB_01_PH" )
   END_RUNG
   RUNG wire#powerrail
      Contact( "Digitais".LSL_002 )
   END_RUNG wire#w1
   RUNG wire#powerrail
      Contact( "Digitais"."LIT_001-YLL" )
   END_RUNG wire#w1
   // the same network as SCL:
   "MB_01_PH" := ("VARIAVEIS".LIT_001 <= "SETPOINTS".SP_NVL_MIN) OR "Digitais".LSL_002 OR "Digitais"."LIT_001-YLL";
END_REGION
END_FUNCTION

FUNCTION_BLOCK "PDIR"   // FB207, LAD
{ S7_Optimized_Access := 'FALSE' }
VERSION : 0.1
// stored: AutoNumber false, IsIECCheckEnabled false, SetENOAutomatically false, UDAEnableTagReadback false
   VAR_INPUT
      ML : Bool;
      MR : Bool;
      DL : Bool;
      MF1 : Bool;
      MF2 : Bool;
      HM : Bool;
      HA : Bool;
      CMA : Bool;
      CLM : Bool;
      CDM : Bool;
      CRF : Bool;
      CRTO : Bool;
      CL1S : Bool;
   END_VAR
   VAR_OUTPUT
      YFPP : Bool;
      YF : Bool;
      CL : Bool;
   END_VAR
   VAR_IN_OUT
      SEG : Int;
      MIN : Int;
      HOR : Int;
   END_VAR
   VAR DB_SPECIFIC
      AUX01 : Bool;
      AUX02 : Bool;
      AUX03 : Bool;
      AUX04 : Bool;
      AUX05 : Bool;
      AUX06 : Bool;
      AUX07 : Bool;
      AUX08 : Bool;
      AUX09 : Bool;
      P60S : Bool;
      P60M : Bool;
      PFHO : Bool;
      TPP1 { S7_SetPoint := 'True'} : TON_TIME;
      TPP2 { S7_SetPoint := 'True'} : TON_TIME;
   END_VAR
   VAR_TEMP
      TEMP0 : Bool;
      TEMP1 : Bool;
      ET_TPP1 : Time;
      ET_TPP2 : Time;
   END_VAR
   VAR_TEMP   // added for the SCL form of the ladder/FBD networks
      _w1 : Bool;
      _w2 : Bool;
      _w3 : Bool;
      _w4 : Bool;
   END_VAR
BEGIN

REGION Network 1: Falha na partida
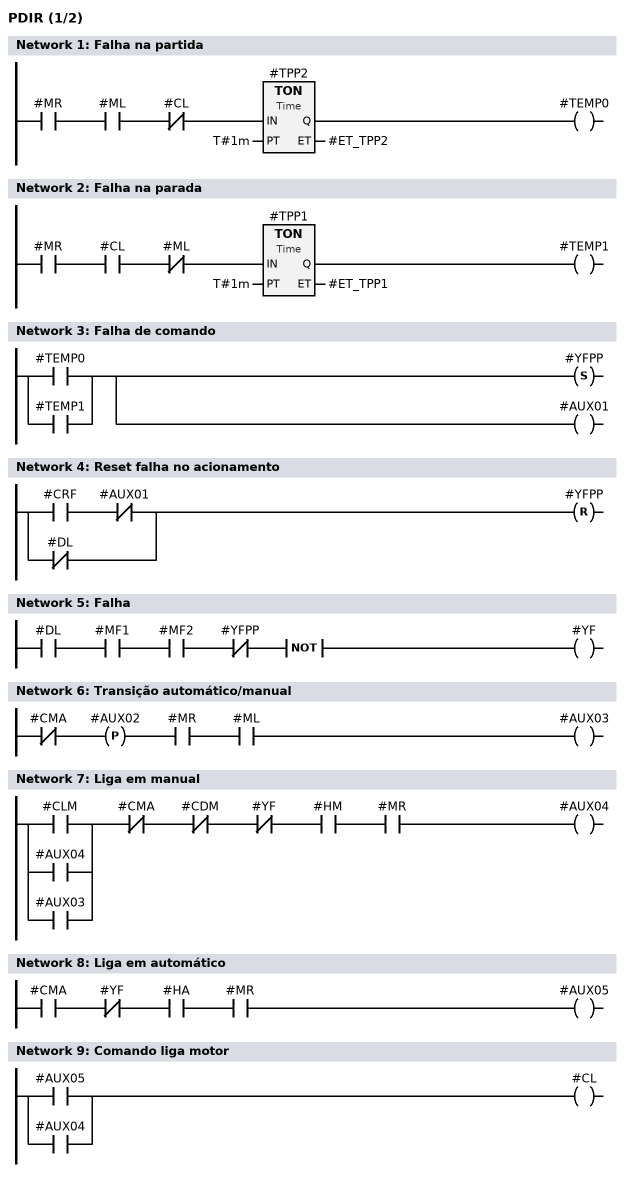
   RUNG wire#powerrail
      Contact( #MR )
      Contact( #ML )
      I_Contact( #CL )
      { S7_Templates := "time_type := Time" } #TPP2.TON(pt := T#1m, et => #ET_TPP2)
      Coil( #TEMP0 )
   END_RUNG
   // the same network as SCL:
   #TPP2(IN := #MR AND #ML AND NOT #CL, PT := T#1m, ET => #ET_TPP2);   // TON
   #TEMP0 := #TPP2.Q;
END_REGION

REGION Network 2: Falha na parada
   RUNG wire#powerrail
      Contact( #MR )
      Contact( #CL )
      I_Contact( #ML )
      { S7_Templates := "time_type := Time" } #TPP1.TON(pt := T#1m, et => #ET_TPP1)
      Coil( #TEMP1 )
   END_RUNG
   // the same network as SCL:
   #TPP1(IN := #MR AND #CL AND NOT #ML, PT := T#1m, ET => #ET_TPP1);   // TON
   #TEMP1 := #TPP1.Q;
END_REGION

REGION Network 3: Falha de comando
   RUNG wire#powerrail
      Contact( #TEMP0 )
      wire#w1
      S_Coil( #YFPP )
   END_RUNG
   RUNG wire#powerrail
      Contact( #TEMP1 )
   END_RUNG wire#w1
   RUNG wire#w1
      Coil( #AUX01 )
   END_RUNG
   // the same network as SCL:
   #_w1 := #TEMP0 OR #TEMP1;
   IF #_w1 THEN #YFPP := TRUE; END_IF;
   #AUX01 := #_w1;
END_REGION

REGION Network 4: Reset falha no acionamento
   RUNG wire#powerrail
      Contact( #CRF )
      I_Contact( #AUX01 )
      wire#w1
      R_Coil( #YFPP )
   END_RUNG
   RUNG wire#powerrail
      I_Contact( #DL )
   END_RUNG wire#w1
   // the same network as SCL:
   IF (#CRF AND NOT #AUX01) OR NOT #DL THEN #YFPP := FALSE; END_IF;
END_REGION

REGION Network 5: Falha
   RUNG wire#powerrail
      Contact( #DL )
      Contact( #MF1 )
      Contact( #MF2 )
      I_Contact( #YFPP )
      Not()
      Coil( #YF )
   END_RUNG
   // the same network as SCL:
   #YF := NOT (#DL AND #MF1 AND #MF2 AND NOT #YFPP);
END_REGION

REGION Network 6: Transição automático/manual
   RUNG wire#powerrail
      I_Contact( #CMA )
      P_Trig( #AUX02 )
      Contact( #MR )
      Contact( #ML )
      Coil( #AUX03 )
   END_RUNG
   // the same network as SCL:
   #_w1 := NOT #CMA AND NOT #AUX02;   // rising edge
   #AUX02 := NOT #CMA;
   #AUX03 := #_w1 AND #MR AND #ML;
END_REGION

REGION Network 7: Liga em manual
   RUNG wire#powerrail
      Contact( #CLM )
      wire#w1
      I_Contact( #CMA )
      I_Contact( #CDM )
      I_Contact( #YF )
      Contact( #HM )
      Contact( #MR )
      Coil( #AUX04 )
   END_RUNG
   RUNG wire#powerrail
      Contact( #AUX04 )
   END_RUNG wire#w1
   RUNG wire#powerrail
      Contact( #AUX03 )
   END_RUNG wire#w1
   // the same network as SCL:
   #AUX04 := (#CLM OR #AUX04 OR #AUX03) AND NOT #CMA AND NOT #CDM AND NOT #YF AND #HM AND #MR;
END_REGION

REGION Network 8: Liga em automático
   RUNG wire#powerrail
      Contact( #CMA )
      I_Contact( #YF )
      Contact( #HA )
      Contact( #MR )
      Coil( #AUX05 )
   END_RUNG
   // the same network as SCL:
   #AUX05 := #CMA AND NOT #YF AND #HA AND #MR;
END_REGION

REGION Network 9: Comando liga motor
   RUNG wire#powerrail
      Contact( #AUX05 )
      wire#w1
      Coil( #CL )
   END_RUNG
   RUNG wire#powerrail
      Contact( #AUX04 )
   END_RUNG wire#w1
   // the same network as SCL:
   #CL := #AUX05 OR #AUX04;
END_REGION

REGION Network 10
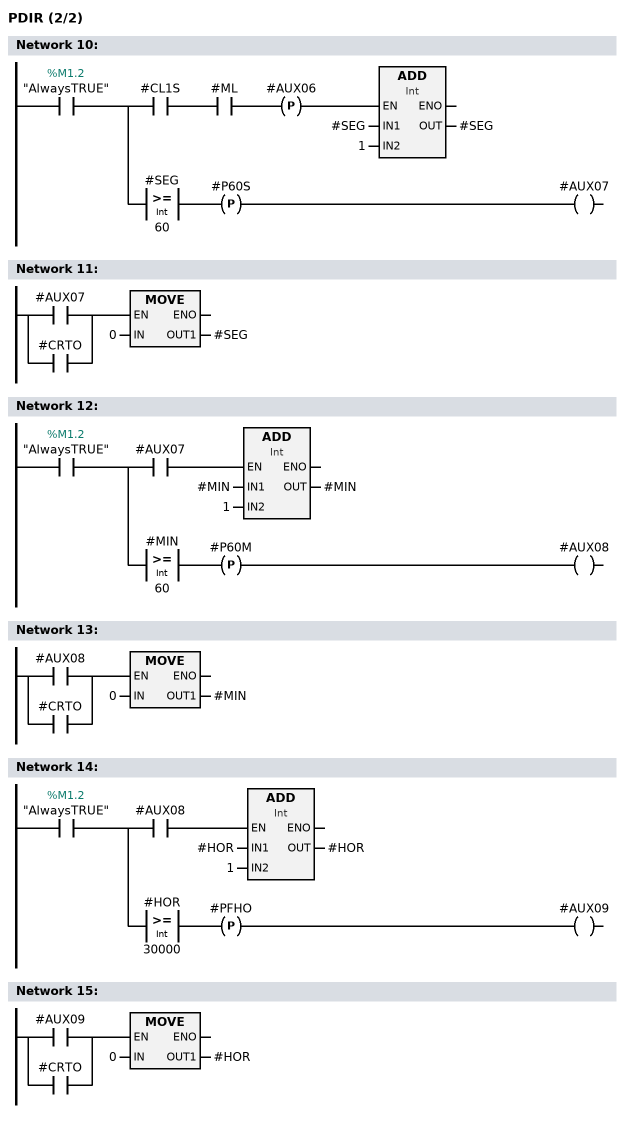
   RUNG wire#powerrail
      Contact( "AlwaysTRUE" )
      wire#w1
      Contact( #CL1S )
      Contact( #ML )
      P_Trig( #AUX06 )
      { S7_Templates := "SrcType := Int"; S7_GenerateENO := "TRUE" } Add(in1 := #SEG, in2 := 1, out => #SEG)
   END_RUNG
   RUNG wire#w1
      { S7_Templates := "SrcType := Int" } GE_Contact(in1 := #SEG, in2 := 60)
      P_Trig( #P60S )
      Coil( #AUX07 )
   END_RUNG
   // the same network as SCL:
   #_w1 := "AlwaysTRUE" AND #CL1S AND #ML;
   #_w2 := #_w1 AND NOT #AUX06;   // rising edge
   #AUX06 := #_w1;
   IF #_w2 THEN #SEG := #SEG + 1; END_IF;
   #_w3 := "AlwaysTRUE" AND (#SEG >= 60);
   #_w4 := #_w3 AND NOT #P60S;   // rising edge
   #P60S := #_w3;
   #AUX07 := #_w4;
END_REGION

REGION Network 11
   RUNG wire#powerrail
      Contact( #AUX07 )
      wire#w1
      { S7_GenerateENO := "TRUE" } Move(in := 0, out1 => #SEG)
   END_RUNG
   RUNG wire#powerrail
      Contact( #CRTO )
   END_RUNG wire#w1
   // the same network as SCL:
   IF #AUX07 OR #CRTO THEN #SEG := 0; END_IF;
END_REGION

REGION Network 12
   RUNG wire#powerrail
      Contact( "AlwaysTRUE" )
      wire#w1
      Contact( #AUX07 )
      { S7_Templates := "SrcType := Int"; S7_GenerateENO := "TRUE" } Add(in1 := #MIN, in2 := 1, out => #MIN)
   END_RUNG
   RUNG wire#w1
      { S7_Templates := "SrcType := Int" } GE_Contact(in1 := #MIN, in2 := 60)
      P_Trig( #P60M )
      Coil( #AUX08 )
   END_RUNG
   // the same network as SCL:
   IF "AlwaysTRUE" AND #AUX07 THEN #MIN := #MIN + 1; END_IF;
   #_w1 := "AlwaysTRUE" AND (#MIN >= 60);
   #_w2 := #_w1 AND NOT #P60M;   // rising edge
   #P60M := #_w1;
   #AUX08 := #_w2;
END_REGION

REGION Network 13
   RUNG wire#powerrail
      Contact( #AUX08 )
      wire#w1
      { S7_GenerateENO := "TRUE" } Move(in := 0, out1 => #MIN)
   END_RUNG
   RUNG wire#powerrail
      Contact( #CRTO )
   END_RUNG wire#w1
   // the same network as SCL:
   IF #AUX08 OR #CRTO THEN #MIN := 0; END_IF;
END_REGION

REGION Network 14
   RUNG wire#powerrail
      Contact( "AlwaysTRUE" )
      wire#w1
      Contact( #AUX08 )
      { S7_Templates := "SrcType := Int"; S7_GenerateENO := "TRUE" } Add(in1 := #HOR, in2 := 1, out => #HOR)
   END_RUNG
   RUNG wire#w1
      { S7_Templates := "SrcType := Int" } GE_Contact(in1 := #HOR, in2 := 30000)
      P_Trig( #PFHO )
      Coil( #AUX09 )
   END_RUNG
   // the same network as SCL:
   IF "AlwaysTRUE" AND #AUX08 THEN #HOR := #HOR + 1; END_IF;
   #_w1 := "AlwaysTRUE" AND (#HOR >= 30000);
   #_w2 := #_w1 AND NOT #PFHO;   // rising edge
   #PFHO := #_w1;
   #AUX09 := #_w2;
END_REGION

REGION Network 15
   RUNG wire#powerrail
      Contact( #AUX09 )
      wire#w1
      { S7_GenerateENO := "TRUE" } Move(in := 0, out1 => #HOR)
   END_RUNG
   RUNG wire#powerrail
      Contact( #CRTO )
   END_RUNG wire#w1
   // the same network as SCL:
   IF #AUX09 OR #CRTO THEN #HOR := 0; END_IF;
END_REGION
END_FUNCTION_BLOCK

FUNCTION "MB-02" : Void   // FC23, LAD
TITLE = Lógica de acionamento do motor
{ S7_Optimized_Access := 'FALSE' }
VERSION : 0.1
// stored: AutoNumber false, IsIECCheckEnabled false, SetENOAutomatically false, UDAEnableTagReadback false
   VAR_TEMP
      IM : Bool;   // Intertravamento manual = 0
      IA : Bool;   // Intertravamento automáticol = 0
      HABM : Bool;   // Habilita funcionamento manual = 1
      HABA : Bool;   // Habilita funcionamento automático = 1
      CLM : Bool;   // Comando liga motor
      PROT : Bool;   // Proteção do motor acionada
   END_VAR
BEGIN

REGION Network 1: Intertravamento maual/automático
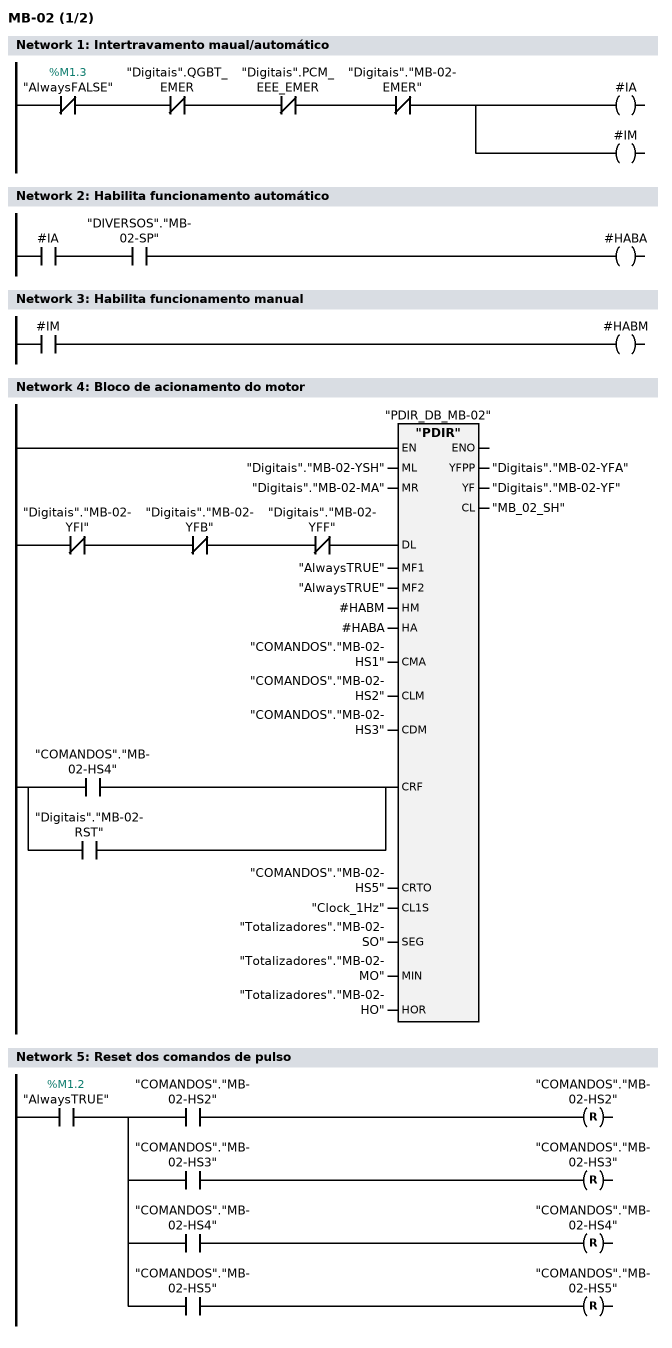
   RUNG wire#powerrail
      I_Contact( "AlwaysFALSE" )
      I_Contact( "Digitais".QGBT_EMER )
      I_Contact( "Digitais".PCM_EEE_EMER )
      I_Contact( "Digitais"."MB-02-EMER" )
      wire#w1
      Coil( #IA )
   END_RUNG
   RUNG wire#w1
      Coil( #IM )
   END_RUNG
   // the same network as SCL:
   #IA := NOT "AlwaysFALSE" AND NOT "Digitais".QGBT_EMER AND NOT "Digitais".PCM_EEE_EMER AND NOT "Digitais"."MB-02-EMER";
   #IM := #IA;
END_REGION

REGION Network 2: Habilita funcionamento automático
   RUNG wire#powerrail
      Contact( #IA )
      Contact( "DIVERSOS"."MB-02-SP" )
      Coil( #HABA )
   END_RUNG
   // the same network as SCL:
   #HABA := #IA AND "DIVERSOS"."MB-02-SP";
END_REGION

REGION Network 3: Habilita funcionamento manual
   RUNG wire#powerrail
      Contact( #IM )
      Coil( #HABM )
   END_RUNG
   // the same network as SCL:
   #HABM := #IM;
END_REGION

REGION Network 4: Bloco de acionamento do motor
   RUNG wire#powerrail
      "PDIR_DB_MB-02"(DL := wire#w1, CRF := wire#w2, ML := "Digitais"."MB-02-YSH", MR := "Digitais"."MB-02-MA", MF1 := "AlwaysTRUE", MF2 := "AlwaysTRUE", HM := #HABM, HA := #HABA, CMA := "COMANDOS"."MB-02-HS1", CLM := "COMANDOS"."MB-02-HS2", CDM := "COMANDOS"."MB-02-HS3", CRTO := "COMANDOS"."MB-02-HS5", CL1S := "Clock_1Hz", SEG := "Totalizadores"."MB-02-SO", MIN := "Totalizadores"."MB-02-MO", HOR := "Totalizadores"."MB-02-HO", YFPP => "Digitais"."MB-02-YFA", YF => "Digitais"."MB-02-YF", CL => "MB_02_SH")
   END_RUNG
   RUNG wire#powerrail
      I_Contact( "Digitais"."MB-02-YFI" )
      I_Contact( "Digitais"."MB-02-YFB" )
      I_Contact( "Digitais"."MB-02-YFF" )
   END_RUNG wire#w1
   RUNG wire#powerrail
      Contact( "COMANDOS"."MB-02-HS4" )
   END_RUNG wire#w2
   RUNG wire#powerrail
      Contact( "Digitais"."MB-02-RST" )
   END_RUNG wire#w2
   // the same network as SCL:
   "PDIR_DB_MB-02"(ML := "Digitais"."MB-02-YSH",   // "PDIR"
                   MR := "Digitais"."MB-02-MA",
                   DL := NOT "Digitais"."MB-02-YFI" AND NOT "Digitais"."MB-02-YFB" AND NOT "Digitais"."MB-02-YFF",
                   MF1 := "AlwaysTRUE",
                   MF2 := "AlwaysTRUE",
                   HM := #HABM,
                   HA := #HABA,
                   CMA := "COMANDOS"."MB-02-HS1",
                   CLM := "COMANDOS"."MB-02-HS2",
                   CDM := "COMANDOS"."MB-02-HS3",
                   CRF := "COMANDOS"."MB-02-HS4" OR "Digitais"."MB-02-RST",
                   CRTO := "COMANDOS"."MB-02-HS5",
                   CL1S := "Clock_1Hz",
                   SEG := "Totalizadores"."MB-02-SO",
                   MIN := "Totalizadores"."MB-02-MO",
                   HOR := "Totalizadores"."MB-02-HO",
                   YFPP => "Digitais"."MB-02-YFA",
                   YF => "Digitais"."MB-02-YF",
                   CL => "MB_02_SH");
END_REGION

REGION Network 5: Reset dos comandos de pulso
   RUNG wire#powerrail
      Contact( "AlwaysTRUE" )
      wire#w1
      Contact( "COMANDOS"."MB-02-HS2" )
      R_Coil( "COMANDOS"."MB-02-HS2" )
   END_RUNG
   RUNG wire#w1
      Contact( "COMANDOS"."MB-02-HS3" )
      R_Coil( "COMANDOS"."MB-02-HS3" )
   END_RUNG
   RUNG wire#w1
      Contact( "COMANDOS"."MB-02-HS4" )
      R_Coil( "COMANDOS"."MB-02-HS4" )
   END_RUNG
   RUNG wire#w1
      Contact( "COMANDOS"."MB-02-HS5" )
      R_Coil( "COMANDOS"."MB-02-HS5" )
   END_RUNG
   // the same network as SCL:
   IF "AlwaysTRUE" AND "COMANDOS"."MB-02-HS2" THEN "COMANDOS"."MB-02-HS2" := FALSE; END_IF;
   IF "AlwaysTRUE" AND "COMANDOS"."MB-02-HS3" THEN "COMANDOS"."MB-02-HS3" := FALSE; END_IF;
   IF "AlwaysTRUE" AND "COMANDOS"."MB-02-HS4" THEN "COMANDOS"."MB-02-HS4" := FALSE; END_IF;
   IF "AlwaysTRUE" AND "COMANDOS"."MB-02-HS5" THEN "COMANDOS"."MB-02-HS5" := FALSE; END_IF;
END_REGION

REGION Network 6: Elevatoria principal modo automatico
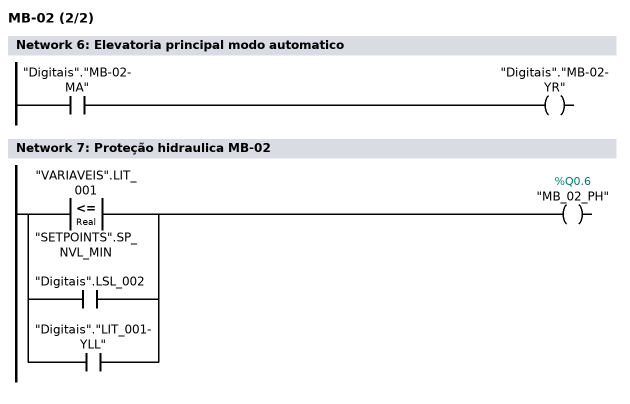
   RUNG wire#powerrail
      Contact( "Digitais"."MB-02-MA" )
      Coil( "Digitais"."MB-02-YR" )
   END_RUNG
   // the same network as SCL:
   "Digitais"."MB-02-YR" := "Digitais"."MB-02-MA";
END_REGION

REGION Network 7: Proteção hidraulica MB-02
   RUNG wire#powerrail
      { S7_Templates := "SrcType := Real" } LE_Contact(in1 := "VARIAVEIS".LIT_001, in2 := "SETPOINTS".SP_NVL_MIN)
      wire#w1
      Coil( "MB_02_PH" )
   END_RUNG
   RUNG wire#powerrail
      Contact( "Digitais".LSL_002 )
   END_RUNG wire#w1
   RUNG wire#powerrail
      Contact( "Digitais"."LIT_001-YLL" )
   END_RUNG wire#w1
   // the same network as SCL:
   "MB_02_PH" := ("VARIAVEIS".LIT_001 <= "SETPOINTS".SP_NVL_MIN) OR "Digitais".LSL_002 OR "Digitais"."LIT_001-YLL";
END_REGION
END_FUNCTION

FUNCTION "MB-03" : Void   // FC24, LAD
TITLE = Lógica de acionamento do motor
{ S7_Optimized_Access := 'FALSE' }
VERSION : 0.1
// stored: AutoNumber false, IsIECCheckEnabled false, SetENOAutomatically false, UDAEnableTagReadback false
   VAR_TEMP
      IM : Bool;   // Intertravamento manual = 0
      IA : Bool;   // Intertravamento automáticol = 0
      HABM : Bool;   // Habilita funcionamento manual = 1
      HABA : Bool;   // Habilita funcionamento automático = 1
      CLM : Bool;   // Comando liga motor
      PROT : Bool;   // Proteção do motor acionada
   END_VAR
BEGIN

REGION Network 1: Intertravamento maual/automático
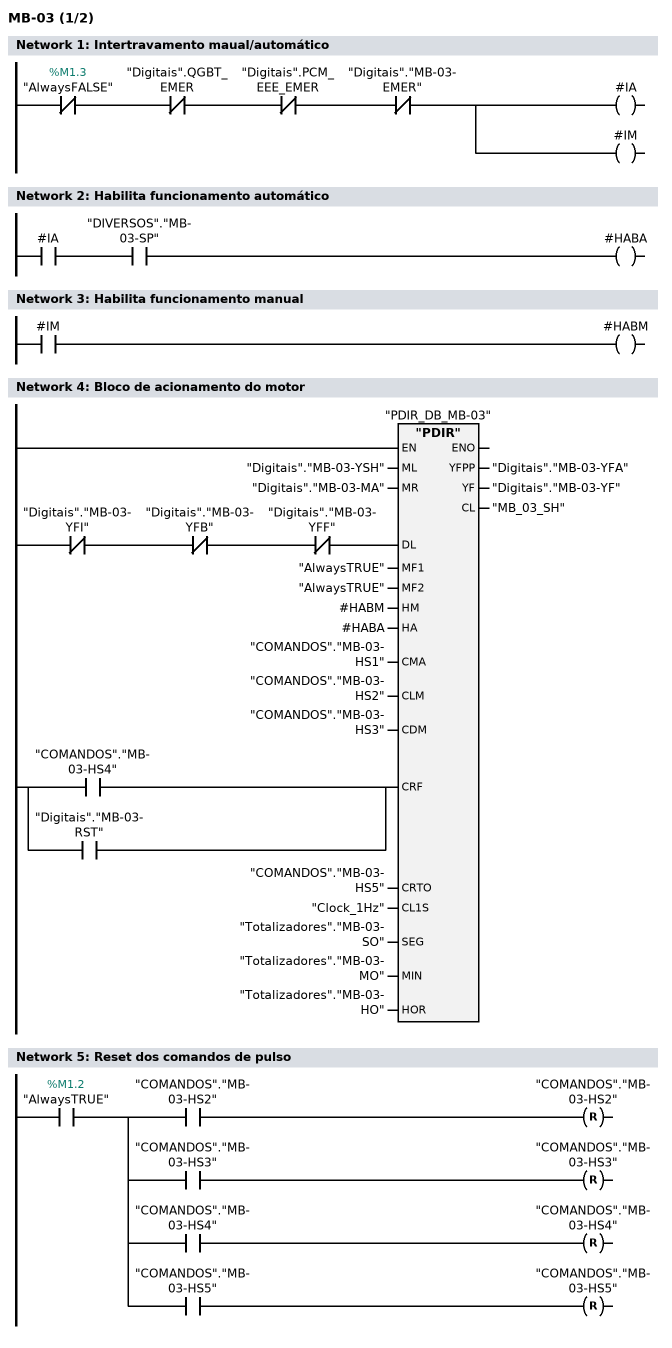
   RUNG wire#powerrail
      I_Contact( "AlwaysFALSE" )
      I_Contact( "Digitais".QGBT_EMER )
      I_Contact( "Digitais".PCM_EEE_EMER )
      I_Contact( "Digitais"."MB-03-EMER" )
      wire#w1
      Coil( #IA )
   END_RUNG
   RUNG wire#w1
      Coil( #IM )
   END_RUNG
   // the same network as SCL:
   #IA := NOT "AlwaysFALSE" AND NOT "Digitais".QGBT_EMER AND NOT "Digitais".PCM_EEE_EMER AND NOT "Digitais"."MB-03-EMER";
   #IM := #IA;
END_REGION

REGION Network 2: Habilita funcionamento automático
   RUNG wire#powerrail
      Contact( #IA )
      Contact( "DIVERSOS"."MB-03-SP" )
      Coil( #HABA )
   END_RUNG
   // the same network as SCL:
   #HABA := #IA AND "DIVERSOS"."MB-03-SP";
END_REGION

REGION Network 3: Habilita funcionamento manual
   RUNG wire#powerrail
      Contact( #IM )
      Coil( #HABM )
   END_RUNG
   // the same network as SCL:
   #HABM := #IM;
END_REGION

REGION Network 4: Bloco de acionamento do motor
   RUNG wire#powerrail
      "PDIR_DB_MB-03"(DL := wire#w1, CRF := wire#w2, ML := "Digitais"."MB-03-YSH", MR := "Digitais"."MB-03-MA", MF1 := "AlwaysTRUE", MF2 := "AlwaysTRUE", HM := #HABM, HA := #HABA, CMA := "COMANDOS"."MB-03-HS1", CLM := "COMANDOS"."MB-03-HS2", CDM := "COMANDOS"."MB-03-HS3", CRTO := "COMANDOS"."MB-03-HS5", CL1S := "Clock_1Hz", SEG := "Totalizadores"."MB-03-SO", MIN := "Totalizadores"."MB-03-MO", HOR := "Totalizadores"."MB-03-HO", YFPP => "Digitais"."MB-03-YFA", YF => "Digitais"."MB-03-YF", CL => "MB_03_SH")
   END_RUNG
   RUNG wire#powerrail
      I_Contact( "Digitais"."MB-03-YFI" )
      I_Contact( "Digitais"."MB-03-YFB" )
      I_Contact( "Digitais"."MB-03-YFF" )
   END_RUNG wire#w1
   RUNG wire#powerrail
      Contact( "COMANDOS"."MB-03-HS4" )
   END_RUNG wire#w2
   RUNG wire#powerrail
      Contact( "Digitais"."MB-03-RST" )
   END_RUNG wire#w2
   // the same network as SCL:
   "PDIR_DB_MB-03"(ML := "Digitais"."MB-03-YSH",   // "PDIR"
                   MR := "Digitais"."MB-03-MA",
                   DL := NOT "Digitais"."MB-03-YFI" AND NOT "Digitais"."MB-03-YFB" AND NOT "Digitais"."MB-03-YFF",
                   MF1 := "AlwaysTRUE",
                   MF2 := "AlwaysTRUE",
                   HM := #HABM,
                   HA := #HABA,
                   CMA := "COMANDOS"."MB-03-HS1",
                   CLM := "COMANDOS"."MB-03-HS2",
                   CDM := "COMANDOS"."MB-03-HS3",
                   CRF := "COMANDOS"."MB-03-HS4" OR "Digitais"."MB-03-RST",
                   CRTO := "COMANDOS"."MB-03-HS5",
                   CL1S := "Clock_1Hz",
                   SEG := "Totalizadores"."MB-03-SO",
                   MIN := "Totalizadores"."MB-03-MO",
                   HOR := "Totalizadores"."MB-03-HO",
                   YFPP => "Digitais"."MB-03-YFA",
                   YF => "Digitais"."MB-03-YF",
                   CL => "MB_03_SH");
END_REGION

REGION Network 5: Reset dos comandos de pulso
   RUNG wire#powerrail
      Contact( "AlwaysTRUE" )
      wire#w1
      Contact( "COMANDOS"."MB-03-HS2" )
      R_Coil( "COMANDOS"."MB-03-HS2" )
   END_RUNG
   RUNG wire#w1
      Contact( "COMANDOS"."MB-03-HS3" )
      R_Coil( "COMANDOS"."MB-03-HS3" )
   END_RUNG
   RUNG wire#w1
      Contact( "COMANDOS"."MB-03-HS4" )
      R_Coil( "COMANDOS"."MB-03-HS4" )
   END_RUNG
   RUNG wire#w1
      Contact( "COMANDOS"."MB-03-HS5" )
      R_Coil( "COMANDOS"."MB-03-HS5" )
   END_RUNG
   // the same network as SCL:
   IF "AlwaysTRUE" AND "COMANDOS"."MB-03-HS2" THEN "COMANDOS"."MB-03-HS2" := FALSE; END_IF;
   IF "AlwaysTRUE" AND "COMANDOS"."MB-03-HS3" THEN "COMANDOS"."MB-03-HS3" := FALSE; END_IF;
   IF "AlwaysTRUE" AND "COMANDOS"."MB-03-HS4" THEN "COMANDOS"."MB-03-HS4" := FALSE; END_IF;
   IF "AlwaysTRUE" AND "COMANDOS"."MB-03-HS5" THEN "COMANDOS"."MB-03-HS5" := FALSE; END_IF;
END_REGION

REGION Network 6: Elevatoria principal modo automatico
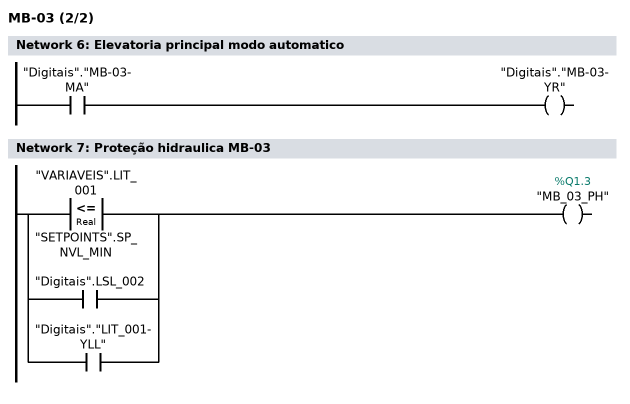
   RUNG wire#powerrail
      Contact( "Digitais"."MB-03-MA" )
      Coil( "Digitais"."MB-03-YR" )
   END_RUNG
   // the same network as SCL:
   "Digitais"."MB-03-YR" := "Digitais"."MB-03-MA";
END_REGION

REGION Network 7: Proteção hidraulica MB-03
   RUNG wire#powerrail
      { S7_Templates := "SrcType := Real" } LE_Contact(in1 := "VARIAVEIS".LIT_001, in2 := "SETPOINTS".SP_NVL_MIN)
      wire#w1
      Coil( "MB_03_PH" )
   END_RUNG
   RUNG wire#powerrail
      Contact( "Digitais".LSL_002 )
   END_RUNG wire#w1
   RUNG wire#powerrail
      Contact( "Digitais"."LIT_001-YLL" )
   END_RUNG wire#w1
   // the same network as SCL:
   "MB_03_PH" := ("VARIAVEIS".LIT_001 <= "SETPOINTS".SP_NVL_MIN) OR "Digitais".LSL_002 OR "Digitais"."LIT_001-YLL";
END_REGION
END_FUNCTION

FUNCTION "MB-04" : Void   // FC25, LAD
TITLE = Lógica de acionamento do motor
{ S7_Optimized_Access := 'FALSE' }
VERSION : 0.1
// stored: AutoNumber false, IsIECCheckEnabled false, SetENOAutomatically false, UDAEnableTagReadback false
   VAR_TEMP
      IM : Bool;   // Intertravamento manual = 0
      IA : Bool;   // Intertravamento automáticol = 0
      HABM : Bool;   // Habilita funcionamento manual = 1
      HABA : Bool;   // Habilita funcionamento automático = 1
      CLM : Bool;   // Comando liga motor
      PROT : Bool;   // Proteção do motor acionada
   END_VAR
BEGIN

REGION Network 1: Intertravamento maual/automático
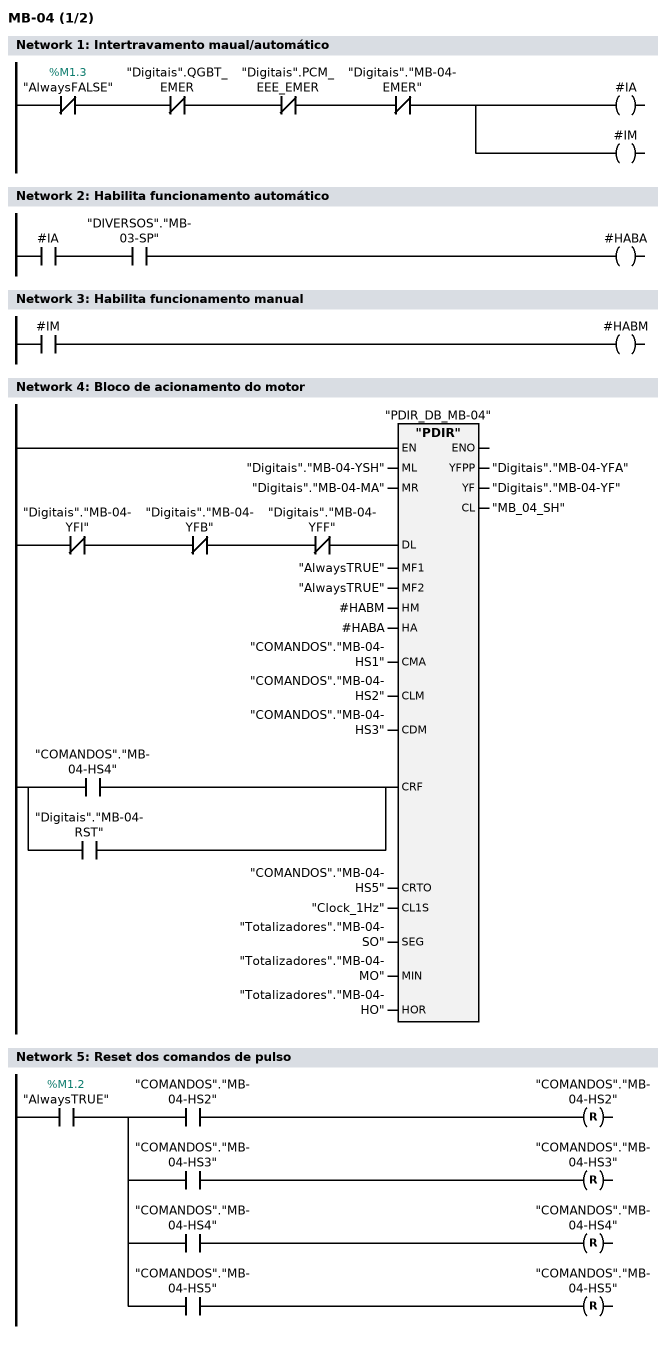
   RUNG wire#powerrail
      I_Contact( "AlwaysFALSE" )
      I_Contact( "Digitais".QGBT_EMER )
      I_Contact( "Digitais".PCM_EEE_EMER )
      I_Contact( "Digitais"."MB-04-EMER" )
      wire#w1
      Coil( #IA )
   END_RUNG
   RUNG wire#w1
      Coil( #IM )
   END_RUNG
   // the same network as SCL:
   #IA := NOT "AlwaysFALSE" AND NOT "Digitais".QGBT_EMER AND NOT "Digitais".PCM_EEE_EMER AND NOT "Digitais"."MB-04-EMER";
   #IM := #IA;
END_REGION

REGION Network 2: Habilita funcionamento automático
   RUNG wire#powerrail
      Contact( #IA )
      Contact( "DIVERSOS"."MB-03-SP" )
      Coil( #HABA )
   END_RUNG
   // the same network as SCL:
   #HABA := #IA AND "DIVERSOS"."MB-03-SP";
END_REGION

REGION Network 3: Habilita funcionamento manual
   RUNG wire#powerrail
      Contact( #IM )
      Coil( #HABM )
   END_RUNG
   // the same network as SCL:
   #HABM := #IM;
END_REGION

REGION Network 4: Bloco de acionamento do motor
   RUNG wire#powerrail
      "PDIR_DB_MB-04"(DL := wire#w1, CRF := wire#w2, ML := "Digitais"."MB-04-YSH", MR := "Digitais"."MB-04-MA", MF1 := "AlwaysTRUE", MF2 := "AlwaysTRUE", HM := #HABM, HA := #HABA, CMA := "COMANDOS"."MB-04-HS1", CLM := "COMANDOS"."MB-04-HS2", CDM := "COMANDOS"."MB-04-HS3", CRTO := "COMANDOS"."MB-04-HS5", CL1S := "Clock_1Hz", SEG := "Totalizadores"."MB-04-SO", MIN := "Totalizadores"."MB-04-MO", HOR := "Totalizadores"."MB-04-HO", YFPP => "Digitais"."MB-04-YFA", YF => "Digitais"."MB-04-YF", CL => "MB_04_SH")
   END_RUNG
   RUNG wire#powerrail
      I_Contact( "Digitais"."MB-04-YFI" )
      I_Contact( "Digitais"."MB-04-YFB" )
      I_Contact( "Digitais"."MB-04-YFF" )
   END_RUNG wire#w1
   RUNG wire#powerrail
      Contact( "COMANDOS"."MB-04-HS4" )
   END_RUNG wire#w2
   RUNG wire#powerrail
      Contact( "Digitais"."MB-04-RST" )
   END_RUNG wire#w2
   // the same network as SCL:
   "PDIR_DB_MB-04"(ML := "Digitais"."MB-04-YSH",   // "PDIR"
                   MR := "Digitais"."MB-04-MA",
                   DL := NOT "Digitais"."MB-04-YFI" AND NOT "Digitais"."MB-04-YFB" AND NOT "Digitais"."MB-04-YFF",
                   MF1 := "AlwaysTRUE",
                   MF2 := "AlwaysTRUE",
                   HM := #HABM,
                   HA := #HABA,
                   CMA := "COMANDOS"."MB-04-HS1",
                   CLM := "COMANDOS"."MB-04-HS2",
                   CDM := "COMANDOS"."MB-04-HS3",
                   CRF := "COMANDOS"."MB-04-HS4" OR "Digitais"."MB-04-RST",
                   CRTO := "COMANDOS"."MB-04-HS5",
                   CL1S := "Clock_1Hz",
                   SEG := "Totalizadores"."MB-04-SO",
                   MIN := "Totalizadores"."MB-04-MO",
                   HOR := "Totalizadores"."MB-04-HO",
                   YFPP => "Digitais"."MB-04-YFA",
                   YF => "Digitais"."MB-04-YF",
                   CL => "MB_04_SH");
END_REGION

REGION Network 5: Reset dos comandos de pulso
   RUNG wire#powerrail
      Contact( "AlwaysTRUE" )
      wire#w1
      Contact( "COMANDOS"."MB-04-HS2" )
      R_Coil( "COMANDOS"."MB-04-HS2" )
   END_RUNG
   RUNG wire#w1
      Contact( "COMANDOS"."MB-04-HS3" )
      R_Coil( "COMANDOS"."MB-04-HS3" )
   END_RUNG
   RUNG wire#w1
      Contact( "COMANDOS"."MB-04-HS4" )
      R_Coil( "COMANDOS"."MB-04-HS4" )
   END_RUNG
   RUNG wire#w1
      Contact( "COMANDOS"."MB-04-HS5" )
      R_Coil( "COMANDOS"."MB-04-HS5" )
   END_RUNG
   // the same network as SCL:
   IF "AlwaysTRUE" AND "COMANDOS"."MB-04-HS2" THEN "COMANDOS"."MB-04-HS2" := FALSE; END_IF;
   IF "AlwaysTRUE" AND "COMANDOS"."MB-04-HS3" THEN "COMANDOS"."MB-04-HS3" := FALSE; END_IF;
   IF "AlwaysTRUE" AND "COMANDOS"."MB-04-HS4" THEN "COMANDOS"."MB-04-HS4" := FALSE; END_IF;
   IF "AlwaysTRUE" AND "COMANDOS"."MB-04-HS5" THEN "COMANDOS"."MB-04-HS5" := FALSE; END_IF;
END_REGION

REGION Network 6: Elevatoria principal modo automatico
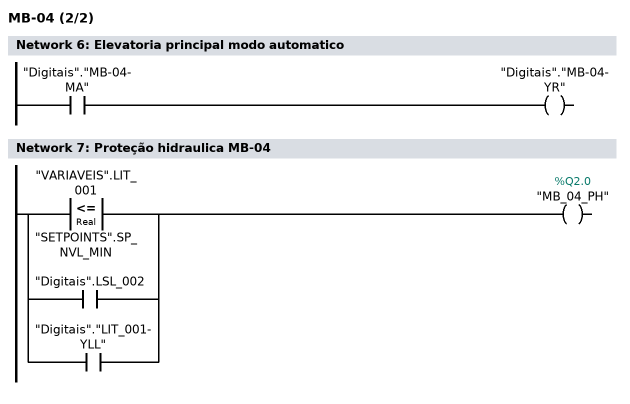
   RUNG wire#powerrail
      Contact( "Digitais"."MB-04-MA" )
      Coil( "Digitais"."MB-04-YR" )
   END_RUNG
   // the same network as SCL:
   "Digitais"."MB-04-YR" := "Digitais"."MB-04-MA";
END_REGION

REGION Network 7: Proteção hidraulica MB-04
   RUNG wire#powerrail
      { S7_Templates := "SrcType := Real" } LE_Contact(in1 := "VARIAVEIS".LIT_001, in2 := "SETPOINTS".SP_NVL_MIN)
      wire#w1
      Coil( "MB_04_PH" )
   END_RUNG
   RUNG wire#powerrail
      Contact( "Digitais".LSL_002 )
   END_RUNG wire#w1
   RUNG wire#powerrail
      Contact( "Digitais"."LIT_001-YLL" )
   END_RUNG wire#w1
   // the same network as SCL:
   "MB_04_PH" := ("VARIAVEIS".LIT_001 <= "SETPOINTS".SP_NVL_MIN) OR "Digitais".LSL_002 OR "Digitais"."LIT_001-YLL";
END_REGION
END_FUNCTION

FUNCTION_BLOCK "ANALOGICOS"   // FB101, LAD
{ S7_Optimized_Access := 'FALSE' }
VERSION : 0.1
// stored: AutoNumber false, IsIECCheckEnabled false, SetENOAutomatically false, UDAEnableTagReadback false
   VAR
      LIT_001 { S7_SetPoint := 'True'} : "INSTRUMENTO";   // Nível Tanque
   END_VAR
BEGIN

REGION Network 1: Nível Tanque (Sensor tipo radar)
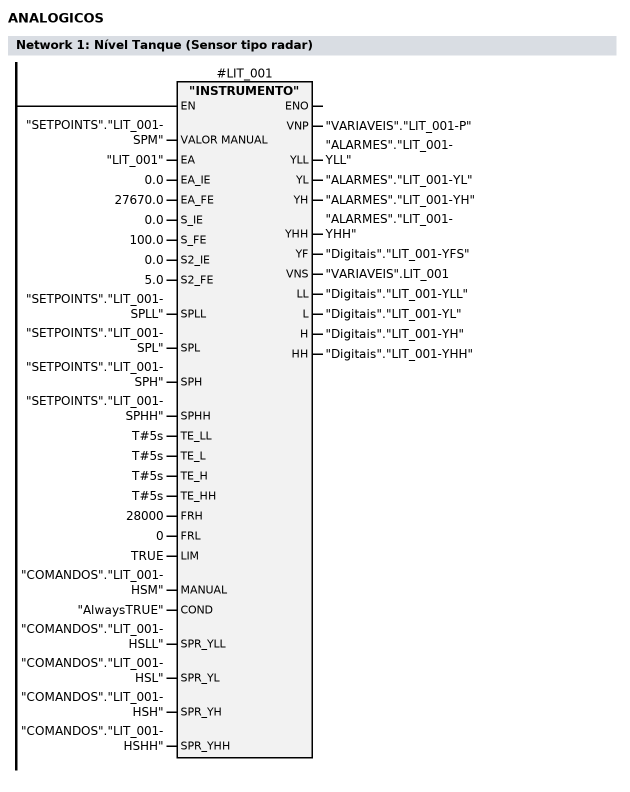
   RUNG wire#powerrail
      #LIT_001("VALOR MANUAL" := "SETPOINTS"."LIT_001-SPM", EA := "LIT_001", EA_IE := 0.0, EA_FE := 27670.0, S_IE := 0.0, S_FE := 100.0, S2_IE := 0.0, S2_FE := 5.0, SPLL := "SETPOINTS"."LIT_001-SPLL", SPL := "SETPOINTS"."LIT_001-SPL", SPH := "SETPOINTS"."LIT_001-SPH", SPHH := "SETPOINTS"."LIT_001-SPHH", TE_LL := T#5s, TE_L := T#5s, TE_H := T#5s, TE_HH := T#5s, FRH := 28000, FRL := 0, LIM := TRUE, MANUAL := "COMANDOS"."LIT_001-HSM", COND := "AlwaysTRUE", SPR_YLL := "COMANDOS"."LIT_001-HSLL", SPR_YL := "COMANDOS"."LIT_001-HSL", SPR_YH := "COMANDOS"."LIT_001-HSH", SPR_YHH := "COMANDOS"."LIT_001-HSHH", VNP => "VARIAVEIS"."LIT_001-P", YLL => "ALARMES"."LIT_001-YLL", YL => "ALARMES"."LIT_001-YL", YH => "ALARMES"."LIT_001-YH", YHH => "ALARMES"."LIT_001-YHH", YF => "Digitais"."LIT_001-YFS", VNS => "VARIAVEIS".LIT_001, LL => "Digitais"."LIT_001-YLL", L => "Digitais"."LIT_001-YL", H => "Digitais"."LIT_001-YH", HH => "Digitais"."LIT_001-YHH")
   END_RUNG
   // the same network as SCL:
   #LIT_001("VALOR MANUAL" := "SETPOINTS"."LIT_001-SPM",   // "INSTRUMENTO"
            EA := "LIT_001",
            EA_IE := 0.0,
            EA_FE := 27670.0,
            S_IE := 0.0,
            S_FE := 100.0,
            S2_IE := 0.0,
            S2_FE := 5.0,
            SPLL := "SETPOINTS"."LIT_001-SPLL",
            SPL := "SETPOINTS"."LIT_001-SPL",
            SPH := "SETPOINTS"."LIT_001-SPH",
            SPHH := "SETPOINTS"."LIT_001-SPHH",
            TE_LL := T#5s,
            TE_L := T#5s,
            TE_H := T#5s,
            TE_HH := T#5s,
            FRH := 28000,
            FRL := 0,
            LIM := TRUE,
            MANUAL := "COMANDOS"."LIT_001-HSM",
            COND := "AlwaysTRUE",
            SPR_YLL := "COMANDOS"."LIT_001-HSLL",
            SPR_YL := "COMANDOS"."LIT_001-HSL",
            SPR_YH := "COMANDOS"."LIT_001-HSH",
            SPR_YHH := "COMANDOS"."LIT_001-HSHH",
            VNP => "VARIAVEIS"."LIT_001-P",
            YLL => "ALARMES"."LIT_001-YLL",
            YL => "ALARMES"."LIT_001-YL",
            YH => "ALARMES"."LIT_001-YH",
            YHH => "ALARMES"."LIT_001-YHH",
            YF => "Digitais"."LIT_001-YFS",
            VNS => "VARIAVEIS".LIT_001,
            LL => "Digitais"."LIT_001-YLL",
            L => "Digitais"."LIT_001-YL",
            H => "Digitais"."LIT_001-YH",
            HH => "Digitais"."LIT_001-YHH");
END_REGION
END_FUNCTION_BLOCK

FUNCTION_BLOCK "INSTRUMENTO"   // FB201, LAD
TITLE = BLOCO PARA CONVERSÃO DE ESCALA DE ENGENHARIA
{ S7_Optimized_Access := 'FALSE' }
VERSION : 0.1
// stored: AutoNumber false, IsIECCheckEnabled false, SetENOAutomatically false, UDAEnableTagReadback false
   VAR_INPUT
      "VALOR MANUAL" : Real;   // VALOR MANUAL (HMI)
      EA : Int;   // LEITURA DO CANAL ANALÓGICO
      EA_IE : Real;   // INÍCIO DA ESCALA DO CANAL
      EA_FE : Real;   // FIM DE ESCALA DO CANAL
      S_IE : Real;   // INÍCIO DE ESCALA DE ENGENHARIA PRINCIPAL
      S_FE : Real;   // FIM DE ESCALA DE ENGENHARIA PRINCIPAL
      S2_IE : Real;   // INÍCIO DE ESCALA DE ENGENHARIA SECUNDÁRIA
      S2_FE : Real;   // FIM DE ESCALA DE ENGENHARIA SECUNDÁRIA
      SPLL : Real;   // SETPOINT MUITO BAIXO
      SPL : Real;   // SETPOINT BAIXO
      SPH : Real;   // SETPOINT ALTO
      SPHH : Real;   // SETPOINT MUITO ALTO
      TE_LL : Time;   // DELAY PARA ALARME MUITO BAIXO
      TE_L : Time;   // DELAY PARA ALARME BAIXO
      TE_H : Time;   // DELAY PARA ALARME ALTO
      TE_HH : Time;   // DELAY PARA ALARME MUITO ALTO
      FRH : Int;   // VALOR ALTO PARA ALARME DE FALHA DE LEITURA
      FRL : Int;   // VALOR BAIXO PARA ALARME DE FALHA DE LEITURA
      LIM : Bool;   // LIMITA O VALOR À ESCALA
      MANUAL : Bool;   // HABILITA MANUTENÇÃO DO INSTRUMENTO
      COND : Bool;   // CONDIÇÃO PARA GERAR ALARME
      SPR_YLL : Bool;   // HABILITA SUPRESSÃO ALARME MUITO BAIXO
      SPR_YL : Bool;   // HABILITA SUPRESSÃO ALARME BAIXO
      SPR_YH : Bool;   // HABILITA SUPRESSÃO ALARME ALTO
      SPR_YHH : Bool;   // HABILITA SUPRESSÃO ALARME MUITO ALTO
   END_VAR
   VAR_OUTPUT
      VNP : Real;   // VALOR CONVERTIDO PARA ESCALA DE ENGENHARIA PRINCIPAL
      YLL : Bool;   // ALARME MUITO BAIXO
      YL : Bool;   // ALARME BAIXO
      YH : Bool;   // ALARME ALTO
      YHH : Bool;   // ALARME MUITO ALTO
      YF : Bool;   // ALARME DE FALHA NA MEDIÇÃO
      VNS : Real;   // VALOR CONVERTIDO PARA ESCALA DE ENGENHARIA SECUNDÁRIA
      LL : Bool;   // VALOR MUITO BAIXO
      L : Bool;   // VALOR BAIXO
      H : Bool;   // VALOR ALTO
      HH : Bool;   // VALOR MUITO ALTO
   END_VAR
   VAR DB_SPECIFIC
      TLL { S7_SetPoint := 'True'} : TON_TIME;   // TEMPO PARA GERAR ALARME
      TL { S7_SetPoint := 'True'} : TON_TIME;   // TEMPO PARA GERAR ALARME
      TH { S7_SetPoint := 'True'} : TON_TIME;   // TEMPO PARA GERAR ALARME
      THH { S7_SetPoint := 'True'} : TON_TIME;   // TEMPO PARA GERAR ALARME
      FALHA : Bool;   // SINALIZAÇÃO DE FALHA NO INSTRUMENTO
   END_VAR
   VAR_TEMP
      EAR : Real;   // VALOR LIDO DA ENTRADA ANALÓGICA
      AC01 : Real;   // AUXILIAR PARA CÁLCULO
      AC02 : Real;   // AUXILIAR PARA CÁLCULO
      AC03 : Real;   // AUXILIAR PARA CÁLCULO
      AC04 : Real;   // AUXILIAR PARA CÁLCULO
      AC05 : Real;   // AUXILIAR PARA CÁLCULO
      AC06 : Real;   // AUXILIAR PARA CÁLCULO
      AC07 : Real;   // AUXILIAR PARA CÁLCULO
      AC08 : Real;   // AUXILIAR PARA CÁLCULO
      AC09 : Real;   // AUXILIAR PARA CÁLCULO
      AC10 : Real;   // AUXILIAR PARA CÁLCULO
      RESULT_P : Real;   // RESULTADO DA ESCALA
      RESULT_S : Real;   // RESULTADO DA ESCALA
      ET_TLL : Time;   // EFETIVO DO TEMPORIZADOR
      ET_TL : Time;   // EFETIVO DO TEMPORIZADOR
      ET_TH : Time;   // EFETIVO DO TEMPORIZADOR
      ET_THH : Time;   // EFETIVO DO TEMPORIZADOR
      EADI : DInt;
   END_VAR
BEGIN

REGION Network 1: CONVERSOR O VALOR LIDO DO CARTÃO PARA REAL
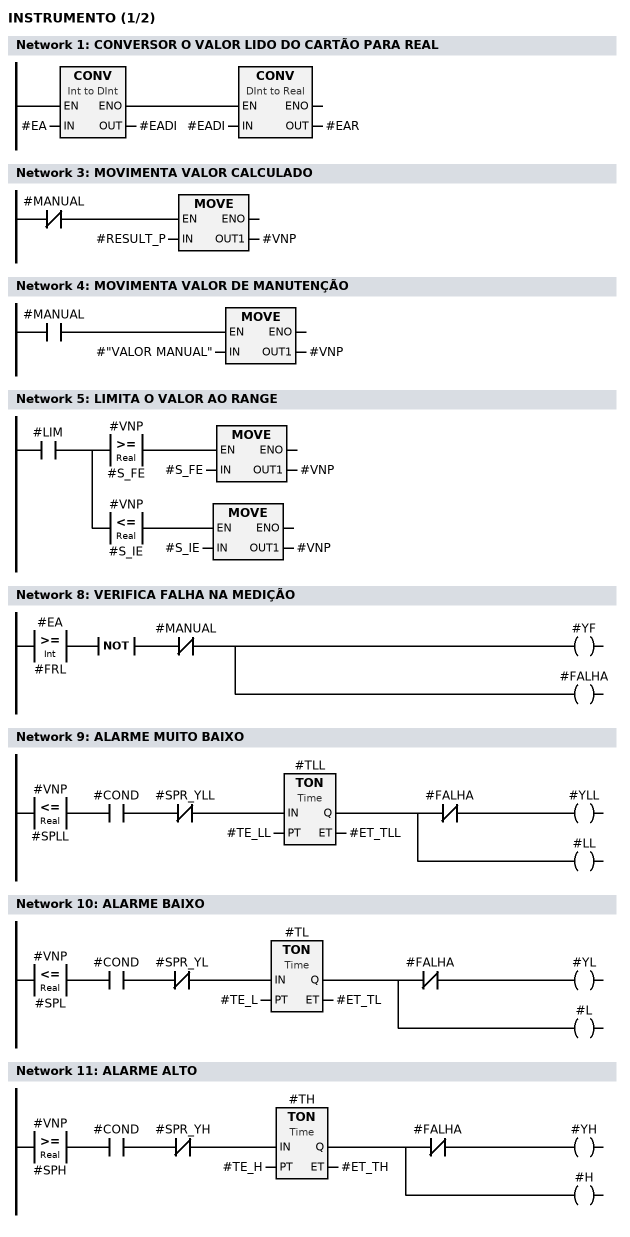
   RUNG wire#powerrail
      { S7_Templates := "[SrcType := Int, DestType := DInt]"; S7_GenerateENO := "TRUE" } Convert(in := #EA, out => #EADI)
      { S7_Templates := "[SrcType := DInt, DestType := Real]"; S7_GenerateENO := "TRUE" } Convert(in := #EADI, out => #EAR)
   END_RUNG
   // the same network as SCL:
   // ENO of a box is taken as its EN; it also drops when the box reports an error
   #EADI := INT_TO_DINT(#EA);
   #EAR := DINT_TO_REAL(#EADI);
END_REGION

NETWORK
TITLE = CONVERTER PARA ESCALA DE ENGENHARIA PRINCIPAL
      L     #EAR;
      L     #EA_IE;
      -R;
      T     #AC01;

      L     #S_FE;  // Subtrai escalas de saída
      L     #S_IE;
      -R;
      T     #AC02;

      L     #EA_FE;  // Subtrai escalas de entrada
      L     #EA_IE;
      -R;
      T     #AC03;

      L     #AC01;  // Multiplica resultado das subtrações
      L     #AC02;
      *R;
      T     #AC04;

      L     #AC04;  // Divide o produto pela subtração das escalas de entrada
      L     #AC03;
      /R;
      T     #AC05;

      L     #AC05;  // Soma o valor de fim da escala de saída
      L     #S_IE;
      +R;
      T     #RESULT_P;  // Resultado do cálculo
      T     #VNP;  // Transfere valor já convertido


REGION Network 3: MOVIMENTA VALOR CALCULADO
   RUNG wire#powerrail
      I_Contact( #MANUAL )
      Move(in := #RESULT_P, out1 => #VNP)
   END_RUNG
   // the same network as SCL:
   IF NOT #MANUAL THEN #VNP := #RESULT_P; END_IF;
END_REGION

REGION Network 4: MOVIMENTA VALOR DE MANUTENÇÃO
   RUNG wire#powerrail
      Contact( #MANUAL )
      Move(in := #"VALOR MANUAL", out1 => #VNP)
   END_RUNG
   // the same network as SCL:
   IF #MANUAL THEN #VNP := #"VALOR MANUAL"; END_IF;
END_REGION

REGION Network 5: LIMITA O VALOR AO RANGE
   RUNG wire#powerrail
      Contact( #LIM )
      wire#w1
      { S7_Templates := "SrcType := Real" } GE_Contact(in1 := #VNP, in2 := #S_FE)
      { S7_GenerateENO := "TRUE" } Move(in := #S_FE, out1 => #VNP)
   END_RUNG
   RUNG wire#w1
      { S7_Templates := "SrcType := Real" } LE_Contact(in1 := #VNP, in2 := #S_IE)
      { S7_GenerateENO := "TRUE" } Move(in := #S_IE, out1 => #VNP)
   END_RUNG
   // the same network as SCL:
   IF #LIM AND (#VNP >= #S_FE) THEN #VNP := #S_FE; END_IF;
   IF #LIM AND (#VNP <= #S_IE) THEN #VNP := #S_IE; END_IF;
END_REGION

NETWORK
TITLE = MOVIMENTA 0 PARA A LEITURA
      A     #YF;
      AN    #MANUAL;
      JNB   _004;
      L     0;
      T     #VNP;
_004: NOP   0;

NETWORK
TITLE = CONVERTER PARA ESCALA DE ENGENHARIA SECUNDÁRIA
      L     #VNP;
      L     #S_IE;
      -R;
      T     #AC06;

      L     #S2_FE;  // Subtrai escalas de saída
      L     #S2_IE;
      -R;
      T     #AC07;

      L     #S_FE;  // Subtrai escalas de entrada
      L     #S_IE;
      -R;
      T     #AC08;

      L     #AC06;  // Multiplica resultado das subtrações
      L     #AC07;
      *R;
      T     #AC09;

      L     #AC09;  // Divide o produto pela subtração das escalas de entrada
      L     #AC08;
      /R;
      T     #AC10;

      L     #AC10;  // Soma o valor de fim da escala de saída
      L     #S2_IE;
      +R;
      T     #RESULT_S;  // Resultado do cálculo
      T     #VNS;  // Transfere valor já convertido


REGION Network 8: VERIFICA FALHA NA MEDIÇÃO
   RUNG wire#powerrail
      { S7_Templates := "SrcType := Int" } GE_Contact(in1 := #EA, in2 := #FRL)
      Not()
      I_Contact( #MANUAL )
      wire#w1
      Coil( #YF )
   END_RUNG
   RUNG wire#w1
      Coil( #FALHA )
   END_RUNG
   // the same network as SCL:
   #YF := NOT (#EA >= #FRL) AND NOT #MANUAL;
   #FALHA := #YF;
END_REGION

REGION Network 9: ALARME MUITO BAIXO
   RUNG wire#powerrail
      { S7_Templates := "SrcType := Real" } LE_Contact(in1 := #VNP, in2 := #SPLL)
      Contact( #COND )
      I_Contact( #SPR_YLL )
      { S7_Templates := "time_type := Time" } #TLL.TON(pt := #TE_LL, et => #ET_TLL)
      wire#w1
      I_Contact( #FALHA )
      Coil( #YLL )
   END_RUNG
   RUNG wire#w1
      Coil( #LL )
   END_RUNG
   // the same network as SCL:
   #TLL(IN := (#VNP <= #SPLL) AND #COND AND NOT #SPR_YLL, PT := #TE_LL, ET => #ET_TLL);   // TON
   #YLL := #TLL.Q AND NOT #FALHA;
   #LL := #TLL.Q;
END_REGION

REGION Network 10: ALARME BAIXO
   RUNG wire#powerrail
      { S7_Templates := "SrcType := Real" } LE_Contact(in1 := #VNP, in2 := #SPL)
      Contact( #COND )
      I_Contact( #SPR_YL )
      { S7_Templates := "time_type := Time" } #TL.TON(pt := #TE_L, et => #ET_TL)
      wire#w1
      I_Contact( #FALHA )
      Coil( #YL )
   END_RUNG
   RUNG wire#w1
      Coil( #L )
   END_RUNG
   // the same network as SCL:
   #TL(IN := (#VNP <= #SPL) AND #COND AND NOT #SPR_YL, PT := #TE_L, ET => #ET_TL);   // TON
   #YL := #TL.Q AND NOT #FALHA;
   #L := #TL.Q;
END_REGION

REGION Network 11: ALARME ALTO
   RUNG wire#powerrail
      { S7_Templates := "SrcType := Real" } GE_Contact(in1 := #VNP, in2 := #SPH)
      Contact( #COND )
      I_Contact( #SPR_YH )
      { S7_Templates := "time_type := Time" } #TH.TON(pt := #TE_H, et => #ET_TH)
      wire#w1
      I_Contact( #FALHA )
      Coil( #YH )
   END_RUNG
   RUNG wire#w1
      Coil( #H )
   END_RUNG
   // the same network as SCL:
   #TH(IN := (#VNP >= #SPH) AND #COND AND NOT #SPR_YH, PT := #TE_H, ET => #ET_TH);   // TON
   #YH := #TH.Q AND NOT #FALHA;
   #H := #TH.Q;
END_REGION

REGION Network 12: ALARME MUITO ALTO
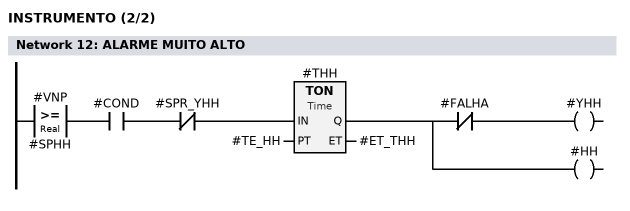
   RUNG wire#powerrail
      { S7_Templates := "SrcType := Real" } GE_Contact(in1 := #VNP, in2 := #SPHH)
      Contact( #COND )
      I_Contact( #SPR_YHH )
      { S7_Templates := "time_type := Time" } #THH.TON(pt := #TE_HH, et => #ET_THH)
      wire#w1
      I_Contact( #FALHA )
      Coil( #YHH )
   END_RUNG
   RUNG wire#w1
      Coil( #HH )
   END_RUNG
   // the same network as SCL:
   #THH(IN := (#VNP >= #SPHH) AND #COND AND NOT #SPR_YHH, PT := #TE_HH, ET => #ET_THH);   // TON
   #YHH := #THH.Q AND NOT #FALHA;
   #HH := #THH.Q;
END_REGION
END_FUNCTION_BLOCK

